(* CODESYS project TcMatrix.library
   DefaultNamespace: TcMatrix
   Description: Matrix arithmatic library
   Author: Andrew Burks
   DocFormat: reStructuredText
   Title: TcMatrix
   Version: 1.4.3
   Company: Burks Engineering
   Placeholder: TcMatrix

Project tree, tasks and I/O mapping:
  libraries: Tc2_Standard, * (Beckhoff Automation GmbH); Tc2_System, * (Beckhoff Automation GmbH); Tc2_Utilities, * (Beckhoff Automation GmbH); Tc3_DynamicMemory, * (Beckhoff Automation GmbH)
  POUs/
    Csv/
      function block MatrixCsvReader [ST]
      function block MatrixCsvWriter [ST]
    Functions/
      Arrays/
        function Array2D_Cols [ST]
        function Array2D_Rows [ST]
        function Array2D_To_Matrix [ST]
        function Matrix_SameSizeAs_Array2D [ST]
        function Matrix_To_Array2D [ST]
      Matrix/
        function Matrix_CanMult [ST]
        function Matrix_Copy [ST]
        function Matrix_DeterminateSquare [ST]
        function Matrix_ElementDifference [ST]
        function Matrix_ElementProduct [ST]
        function Matrix_ElementSum [ST]
        function Matrix_Grow [ST]
        function Matrix_InvertSquare [ST]
        function Matrix_Product [ST]
        function Matrix_Scale [ST]
        function Matrix_Shrink [ST]
        function Matrix_SubMatrix [ST]
        function Matrix_Transpose [ST]
        function Matrix_TransposeSquare [ST]
      Vector/
        function Vector_CrossProduct [ST]
        function Vector_DotProduct [ST]
        function Vector_Magnitude [ST]
        function Vector_Normalize [ST]
    MatrixAccessors/
      function block MatrixAccessor [ST]: Init_, This2Parent, GetI, SetI
      function block ShrunkMatrixAccessor [ST]: Init, Cols, Rows, This2Parent
      function block SubMatrixAccessor [ST]: Init, Cols, Rows, This2Parent
      function block TransposeMatrixAccessor [ST]: Init, Cols, Rows, This2Parent
    function block Array2DStaticMatrix [ST]: GetI, SetI
    function block DynamicMatrix [ST]: LogData, Free, Init, InitArray2D, InitConstant, InitCopy, InitIdentity, InitMagicSquare, InitTrapezoidal, InitVector, InitZeros, Grow, Resize, Shrink, Transpose, Cols, FB_exit, FB_init, GetI, Rows, SetI, AsColVector, AsElementDifference, AsElementProduct, AsElementSum, AsGrown, AsInverse, AsMatrixProduct, AsRowVector, AsScaled, AsShrunk, AsSubMatrix, AsTransposed, AsVectorCrossProduct
    function block ExternalStaticMatrix [ST]: Init, GetI, SetI
    function block Matrix [ST]: GetShrunkMatrixAccessor, GetSubMatrixAccessor, GetTransposeMatrixAccessor, Average, MaxVal, MinVal, Sum, IsEqual, IsEqualSize, IsNearlyEqual, GetDeterminant, GetI, GetRC, GetSize, GetVectorDotProduct, GetVectorMagnitude, CopyTo, GetStringLengthEstimate, IsCleared, IsEmpty, IsNearZero, IsSquare, IsVector, LogError, LogEvent, LogMessage, LogWarning, WriteDataToString, Clear, CopyFrom, ElementDifference, ElementProduct, ElementSum, FillFrom, FillFromArray2D, FillFromAt, FillTrapezoidal, IntPower, InvertSquare, Normalize, Power, Scale, SetI, SetRC, SortByColAsc, SwapI, SwapRC, SwapRow, TransposeSquare, BufferSize, Cols, Length, Rows, sPath, ZeroReference, IC2RC, RC2I, RCC2I
    function block StaticMatrix [ST]: Init_, Cols, Rows
  Version/
    global variables Global_Version
*)

// Version/Global_Version
{attribute 'TcGenerated'}
{attribute 'no-analysis'}
{attribute 'linkalways'}
// This function has been automatically generated from the project information.
VAR_GLOBAL CONSTANT
	{attribute 'const_non_replaced'}
	stLibVersion_TcMatrix : ST_LibVersion := (iMajor := 1, iMinor := 4, iBuild := 3, iRevision := 0, nFlags := 0, sVersion := '1.4.3');
END_VAR

// POUs/Csv/MatrixCsvReader
FUNCTION_BLOCK MatrixCsvReader
VAR_IN_OUT CONSTANT
	M : Matrix;
END_VAR
VAR_INPUT
	bExecute : BOOL;
	sPathName : T_MaxString;
	tTimeout : TIME;//timeout applied indidivudally to each file operation
	nHeaderLines : UDINT;//number of lines to skip at the beginning
END_VAR
VAR_OUTPUT
	bBusy : BOOL;
	bError : BOOL;
	nErrId : UDINT;
	nErrStep : UDINT;
	nRows : UINT;
	nCols : UINT;
	nVals : UINT;
END_VAR
VAR
	FileOpen : FB_FileOpen;
	CsvRead : FB_CSVMemBufferReader;
	FileRead : FB_FileRead;
	FileSeek : FB_FileSeek;
	FileClose : FB_FileClose;
	
	hFile : UINT;
	readEOF : BOOL;
	bytesRead : DINT;
	bytesParsed : DINT;
	buffer : STRING(bufferSize);
	step : UDINT;
	
	Hi : UINT;
	Ri : UINT;
	Ci : UINT;
	BuffCmd : E_EnumCmdType;
END_VAR
VAR CONSTANT
	bufferSize : UDINT := 1024;
	dataSize : UDINT := 16;	

	stepReady : UDINT := 0;
	stepOpenFile : UDINT := 1;
	stepFillBuffer : UDINT := 2;
	stepReadBuffer : UDINT := 3;
	stepMovePointer : UDINT := 4;
	stepCloseFile : UDINT := 5;
	stepDone : UDINT := 6;
END_VAR

FileOpen(
	sNetId := '',
	sPathName := spathname,
	nMode := FOPEN_MODEREAD OR FOPEN_MODEBINARY,
	ePath := E_OpenPath.PATH_GENERIC,
	bExecute := step = stepOpenFile,
	tTimeout := tTimeout);
FileRead(snetId := '',
	hFile := hFile,
	pReadBuff := ADR(buffer),
	cbReadLen := bufferSize,
	bExecute := step = stepFillBuffer,
	tTimeout := tTimeout);
FileSeek(snetID := '',
	hFile := hFile,
	//nSeekPos := 0,
	eOrigin := E_SeekOrigin.SEEK_CUR,
	bExecute := step = stepMovePointer,
	tTimeout := tTimeout);
FileClose(
	snetId := '',
	hFile := hFile,
	bexecute := step = stepCloseFile,
	tTimeout := tTimeout);
			
CASE step OF
	stepReady:
		bError := FALSE;
		nErrId := 0;
		nErrStep := 0;
		
		hFile := 0;
		readEOF := FALSE;
		
		Hi := 0;
		Ri := 0;
		Ci := 0;
		nRows := 0;
		nCols := 0;
		
		IF bExecute THEN
			IF NOT M.IsEmpty THEN
				bBusy := TRUE;
				step := stepOpenFile;
			END_IF
		END_IF
		
	stepOpenFile:
		
		IF FileOpen.bError THEN
			bError := TRUE;
			nErrId := FileOpen.nErrId;
			nErrStep := step;
			step := stepDone;
		ELSIF NOT(FileOpen.bBusy) THEN
			hFile := FileOpen.hFile;
			step := stepFillBuffer;
		END_IF
		
	stepFillBuffer:
		bytesRead := 0;
		IF FileRead.bError THEN
			bError := TRUE;
			nErrId := FileRead.nErrId;
			nErrStep := step;
			step := stepCloseFile;
		ELSIF NOT(FileRead.bBusy) THEN
			bytesRead := UDINT_TO_DINT(FileRead.cbRead);
			readEOF := FileRead.bEOF;//it looks like EOF is mutually exclusive with actually reading bytes. so kind of useless.
			IF bytesRead = 0 THEN
				step := stepCloseFile;
			ELSE
				step := stepReadBuffer;
			END_IF
		END_IF
		
	stepReadBuffer:
		BuffCmd := E_EnumCmdType.eEnumCmd_First;
		bytesParsed := 0;
		REPEAT
			CsvRead(eCmd := BuffCmd,
				pBuffer := ADR(Buffer),
				cbBuffer := DINT_TO_UDINT(bytesRead));
			BuffCmd := E_EnumCmdType.eEnumCmd_Next;
			
			IF CsvRead.bOk THEN
				bytesparsed := bytesparsed + UDINT_TO_DINT(CsvRead.cbRead);
				IF Hi < nHeaderLines THEN
					IF CsvRead.bCRLF THEN
						Hi := Hi + 1;
					END_IF
				ELSE
					IF Ri >= M.Rows OR Ci >= M.Cols THEN
						bError := TRUE;
						nErrId :=1;
						nErrStep := step;
						step := stepCloseFile;
						RETURN;
					END_IF
					M.SetRC(Ri,Ci,STRING_TO_LREAL(CsvRead.getValue));
					Ci := Ci + 1;
					nVals := NVals + 1;
					IF CsvRead.bCRLF THEN
						Ri := Ri + 1;
						Ci := 0;
						nRows := Ri;
					END_IF
					IF Ci > nCols THEN
						nCols := Ci;
					END_IF
				END_IF
			END_IF
		UNTIL
			NOT(CsvRead.bOk)
		END_REPEAT
		IF readEOF THEN//this probably will never happen because EOF seems to be mutually exclusive with reading bytes
			step := stepCloseFile;
		ELSE
			//move pointer backwards to where it was before the read, then forward based on how much data was read from the CSV buffer. This re-reads any partial cells that were not parsed
			FileSeek.nSeekPos := bytesParsed - bytesRead;
			IF FileSeek.nSeekPos <> 0 THEN
				step := stepMovePointer;
			ELSE
				step := stepFillBuffer;
			END_IF;
		END_IF
		
	
		
	stepMovePointer:
		IF FileSeek.bError AND NOT bError THEN
			bError := TRUE;
			nErrId := FileSeek.nErrId;
			nErrStep := step;
			step := stepDone;
		ELSIF NOT(FileSeek.bBusy) THEN
			step := stepFillBuffer;
		END_IF
		
	stepCloseFile:
		
		IF FileClose.bError AND NOT bError THEN
			bError := TRUE;
			nErrId := FileClose.nErrId;
			nErrStep := step;
			step := stepDone;
		ELSIF NOT(FileClose.bBusy) THEN
			step := stepDone;
		END_IF
		
		
	stepDone:
		bBusy := FALSE;
END_CASE

IF NOT bExecute THEN
	step := stepReady;
	bBusy := FALSE;
END_IF

END_FUNCTION_BLOCK

// POUs/Matrix
(*
Matrix Base Class
=============

Overview
-------------

This abstract class encapsulates the logic of manipulating and interacting with matricies without forcing a specific memory management pattern.
Derived classes are:

- DynamicMatrix: A concrete class that dynamically allocates memory to take any form needed
- StaticMatrix: An abstract class that serves as the base for classes with fixed memory sources
- MatrixAccessor: An abstract class that serves as the base for classes that inherit the memory of another matrix and remap it to their own form
 
With either pattern the memory is accessed as a row-major 1D array of LREAL.

*)
{attribute 'reflection'}
{attribute 'no_assign'}
FUNCTION_BLOCK ABSTRACT Matrix
VAR_INPUT
END_VAR
VAR_OUTPUT
END_VAR
VAR

	
	{attribute 'instance-path'}
	{attribute 'noinit'}
	sPath_ : T_MaxString;
	
	Ri : UINT;
	Ci : UINT;
	I : UINT;
	
	ZeroReference_ : LREAL;//numbers below this are considered zero for the purposes of avoiding near-divide-by-zero floating point issues
END_VAR

LogMessage('%s: There is no need to call the main FB function for type Matrix');

METHOD PUBLIC GetShrunkMatrixAccessor : ShrunkMatrixAccessor
VAR_INPUT
	Row : UINT;
	Col : UINT;
END_VAR
GetShrunkMatrixAccessor.Init(THIS^,Row,Col);
END_METHOD

METHOD PUBLIC GetSubMatrixAccessor : SubMatrixAccessor
VAR_INPUT
	RowStart : UINT;
	RowCount : UINT;
	ColStart : UINT;
	ColCount : UINT;
END_VAR
GetSubMatrixAccessor.Init(THIS^,RowStart,RowCount,ColStart,ColCount);
END_METHOD

METHOD PUBLIC GetTransposeMatrixAccessor : TransposeMatrixAccessor
VAR_INPUT
END_VAR
GetTransposeMatrixAccessor.Init(THIS^);
END_METHOD

//returns the average value of all elements
PROPERTY PUBLIC Average : LREAL
GET
IF Length > 0 THEN
	Average := Sum / Length;
ELSE
	Average := 0;
END_IF
END_GET
END_PROPERTY

//Returns the maximum value from all elements
PROPERTY PUBLIC MaxVal : LREAL
GET
VAR
	MaxVal_ : LREAL;
END_VAR
IF IsEmpty THEN
	MaxVal := 0;
ELSE
	MaxVal_ := GetI(0);
	FOR I := 1 TO Length-1 DO
		IF getI(I) < MaxVal_ THEN
			MaxVal_ := GetI(I);
		END_IF
	END_FOR
	MaxVal := MaxVal_;
END_IF
END_GET
END_PROPERTY

//Returns the minimum value from all elements
PROPERTY PUBLIC MinVal : LREAL
GET
VAR
	MinVal_ : LREAL;
END_VAR
IF IsEmpty THEN
	MinVal := 0;
ELSE
	MinVal_ := GetI(0);
	FOR I := 1 TO Length-1 DO
		IF getI(I) < MinVal_ THEN
			MinVal_ := GetI(I);
		END_IF
	END_FOR
	MinVal := MinVal_;
END_IF
END_GET
END_PROPERTY

//Returns the sum of all elements
PROPERTY PUBLIC Sum : LREAL
GET
VAR
	Sum_ : LREAL;
END_VAR
Sum_ := 0;
IF NOT(IsEmpty) THEN
	FOR I := 0 TO Length-1 DO
		Sum_ := Sum_ + GetI(I);
	END_FOR
END_IF
Sum := Sum_;
END_GET
END_PROPERTY

//Determines if this matrix is equal to a supplied matrix.
//
//Two matricies are considered equal if they are the same size and every set of corresponding elements are equal.
//
//.. note:: Two empty matricies are considered equal.
METHOD PUBLIC IsEqual : BOOL//TRUE if the two matricies are equal, FALSE if they are not
VAR_IN_OUT CONSTANT
	M : Matrix;//The other matrix to compare to this one
END_VAR
IF NOT( IsEqualSize(M)) THEN
	IsEqual := FALSE;
	RETURN;
END_IF

//If either matrix is empty don't bother comparing elements
IF IsEmpty OR M.IsEmpty THEN
	//If both are empty then they are equal
	IsEqual := IsEmpty AND M.IsEmpty;
	RETURN;
END_IF

//Both Rows and Cols must be non zero for this loop to not go bonkers
FOR Ri := 0 TO Rows-1 DO
	FOR Ci := 0 TO Cols-1 DO
		IF NOT(GetRC(Ri,Ci) = M.GetRC(Ri,Ci)) THEN
			IsEqual := FALSE;
			RETURN;
		END_IF
	END_FOR
END_FOR

IsEqual := TRUE;
END_METHOD

//Checks if this matrix is the same size (number of rows and number of columns match) as the supplied matrix.
//
//.. note:: two empty matricies are considered the same size.
METHOD PUBLIC IsEqualSize : BOOL//True if this matrix is the same size as the supplied matrix
VAR_IN_OUT CONSTANT
	M : Matrix;//The matrix which should have its size compared to the size of this matrix
END_VAR
IsEqualSize := M.Rows = Rows AND M.Cols = Cols;
END_METHOD

//Determines if this matrix is *nearly* equal to a supplied matrix, based on a supplied precision.
//
//Two matricies are considered nearly equal if they are the same size and every set of corresponding elements are equal to within the supplied precision.
//.. note:: Note that two empty matricies are considered equal
METHOD PUBLIC IsNearlyEqual : BOOL//TRUE if the two matricies are nearly equal, FALSE if they are not
VAR_IN_OUT CONSTANT
	M : Matrix;//The other matrix to compare to this one
END_VAR
VAR_INPUT
	Precision : LREAL;//Deviation between two elements larger than this value makes them unequal
END_VAR
IF NOT( IsEqualSize(M)) THEN
	IsNearlyEqual := FALSE;
	RETURN;
END_IF

//If either matrix is empty don't bother comparing elements
IF IsEmpty OR M.IsEmpty THEN
	//If both are empty then they are equal
	IsNearlyEqual := IsEmpty AND M.IsEmpty;
	RETURN;
END_IF

//Both Rows and Cols must be non zero for this loop to not go bonkers
FOR Ri := 0 TO Rows-1 DO
	FOR Ci := 0 TO Cols-1 DO
		IF NOT( ABS(GetRC(Ri,Ci) - M.GetRC(Ri,Ci)) < Precision) THEN
			IsNearlyEqual := FALSE;
			RETURN;
		END_IF
	END_FOR
END_FOR

IsNearlyEqual := TRUE;
END_METHOD

//Gets the determinant of this matrix
//
//:Prerequisites:
// - Matrix is not empty
// - Matrix is square
//
//.. note:: If this matrix does not meet the requirements 0 is returned
METHOD PUBLIC GetDeterminant : LREAL//The determinant of this matrix, if the prerequisites are met. Otherwise, returns 0.
VAR_INPUT
END_VAR
VAR
	Res : LREAL;
END_VAR
IF NOT(Matrix_DeterminateSquare(M := THIS^,Res => Res)) THEN
	LogWarning('%s: Unable to calculate determinate');
	GetDeterminant := 0;
ELSE
	GetDeterminant := Res;
END_IF
END_METHOD

//Gets the value of the element in this matrix at the supplied location as if the elements were stored in a 1D row-major array
//
//:Prerequisites:
// - I < Rows*Cols
// - Matrix is not empty
//
//.. note:: If the supplied index is out of bounds the value 0 is returned and a warning is generated in the Error List
METHOD PUBLIC ABSTRACT GetI : LREAL//The value of the element at the specified index, or 0 if an invalid index is supplied
VAR_INPUT
	I : UINT;//The index of the element which should have its value returned
END_VAR
END_METHOD

//returns the value of the element of this matrix at the specified row and column.
//
//:Prerequisites:
// - Row < Rows
// - Col < Cols
// - Matrix is not empty
//
//.. note:: If the supplied or or column is out of bounds then a warning message is generated in the Error List and the value 0 is returned
METHOD PUBLIC GetRC : LREAL//The value of the element at the specified row and column, or 0 if an invalid index is supplied
VAR_INPUT
	Row : UINT;//The row of the element to fetch
	Col : UINT;//The column of the element to fetch
END_VAR
IF IsEmpty THEN
	GetRC := 0;
	LogWarning('%s: Attempted RC access of empty Matrix');
ELSIF
	Row >= Rows THEN
	GetRC := 0;
	LogWarning('%s: Attempted RC access of out-of-bound matrix row');
ELSIF
	Col >= Cols THEN
	GetRC := 0;
	LogWarning('%s: Attempted RC access of out-of-bounds Matrix column');
ELSE
	GetRC := GetI(RC2I(Row,Col));
END_IF
END_METHOD

//Returns the length of the matrix in the specified dimension
//
// - GetSize(0) is equivalent to Rows
// - GetSize(1) is equivalent to Cols
//
//.. note:: If an invalid dimension is supplied then a warning is generated in the Error List and the value 0 is returned
METHOD PUBLIC GetSize : UINT//The length of the matrix in the specified dimension, or 0 if the dimension specified is invalid
VAR_INPUT
	Dim : UINT;//The dimension of the matrix for which the size should be returned. 0=Rows, 1=Cols
END_VAR
IF Dim = 0 THEN
	GetSize := Rows;
ELSIF Dim = 1 THEN
	GetSize := Cols;
ELSE
	LogWarning('%s: Attempted to GetSize for a dimension other than 0 or 1');
	GetSize := 0;
END_IF
END_METHOD

//Returns the vector dot product of this matrix and the supplied other matrix (ignoring the orientation of both matricies).
//:Prerequisites:
// - This matrix is a vector and is not empty
// - The supplied other matrix is a vector and is not empty
// - This vector has the same length (but not necessarily orientation) as the supplied vector
METHOD PUBLIC GetVectorDotProduct : LREAL//The dot product (element-wise product) of this vector and the supplied vector, or 0 if the inputs are invalid
VAR_IN_OUT CONSTANT
	V : Matrix;//The vector which which the dot product of this vector should be taken.
END_VAR
VAR
	Res : LREAL;
END_VAR
IF NOT(Vector_DotProduct(V,THIS^,Res => Res)) THEN
	LogWarning('%s: Unable to calculate vector dot product');
	GetVectorDotProduct := 0;
ELSE
	GetVectorDotProduct := Res;
END_IF
END_METHOD

//Calcualtes the vector magnitude of this matrix (square root of the sum of the squares), assuming it is a vector.
//
//:Prerequisites:
// - This matrix is not empty and is a vector
//
//.. note:: If this matrix is empty or is not a vector, 0 is returned
METHOD PUBLIC GetVectorMagnitude : LREAL//The vector magnitude of this matrix if it is a vector, otherwise 0
VAR_INPUT
END_VAR
VAR
	Res : LREAL;
END_VAR
IF NOT(Vector_Magnitude(THIS^,Res => Res)) THEN
	LogWarning('%s: Unable to calculate vector magnitude');
	GetVectorMagnitude := 0;
ELSE
	GetVectorMagnitude := Res;
END_IF
END_METHOD

(*Copy the value from each element in this matrix to each corresponding element in the destination matrix

:Prerequisites:
 - This matrix is the same size as the destination matrix
 - Neither matrix is empty
 
 *)
METHOD PUBLIC CopyTo : BOOL//Returns true if the prerequisites were met and the data was copied, false otherwise
VAR_IN_OUT
	M : Matrix;//Destination for the copy operation
END_VAR
CopyTo := Matrix_Copy(THIS^,M);
END_METHOD

//Calulates how long of a string (in Bytes) is required in order to print the entire contents of the matrix using the WriteDataToString function
METHOD PUBLIC GetStringLengthEstimate : UDINT;
VAR_INPUT
END_VAR
VAR
	CharsPerElement : UDINT := 20;//15 point precision, decimal, sign, leading zero, comma, space
	CharsPerRow : UDINT := 6;//space, semicolon, carriage return, line return, space, space
	CharsPerMatrix : UDINT := 4;//open bracket, space ; space, closing bracket
END_VAR
GetStringLengthEstimate := 1+CharsPerMatrix + CharsPerRow * Rows + CharsPerElement * Length;//extra one for null character
END_METHOD

//Returns TRUE if every element of the matrix is equal to zero, or the matrix is empty
PROPERTY PUBLIC IsCleared : BOOL
GET
IF IsEmpty THEN
	IsCleared := TRUE;
	RETURN;
END_IF

FOR Ri := 0 TO Rows-1 DO
	FOR Ci := 0 TO Cols-1 DO
		IF GetRC(Ri,Ci) <> 0 THEN
			IsCleared := FALSE;
			RETURN;
		END_IF
	END_FOR
END_FOR

IsCleared := TRUE;
END_GET
END_PROPERTY

//Returns true if the matrix does not have any addresible elements
PROPERTY PUBLIC IsEmpty : Bool
GET
IsEmpty := Length = 0;
END_GET
END_PROPERTY

//Returns true if the supplied value is near enough to zero that it should not be used as a divisor. See the property ZeroReference
METHOD PROTECTED IsNearZero : BOOL
VAR_INPUT
	IN : LREAL;//The value which should have its magnitude evaluated
END_VAR
IsNearZero := ABS(IN) < ZeroReference;
END_METHOD

//Returns true if this matrix is not empty, and the number of columns is equal to the number of rows
PROPERTY PUBLIC IsSquare : BOOL
GET
IsSquare := NOT(IsEmpty) AND Rows = Cols;
END_GET
END_PROPERTY

//Returns true if this matrix is not empty, and at least one dimension has a size of 1 (row vector or column vector).
PROPERTY PUBLIC IsVector : BOOL
GET
IsVector := NOT(IsEmpty) AND (Rows = 1) OR (Cols = 1);
END_GET
END_PROPERTY

//Logs the supplied message to the error output as an 'Error'
METHOD PROTECTED LogError
VAR_INPUT
	Message : T_MaxString;//The message to log. %s is substituted with the symbolic address of this matrix.
END_VAR
ADSLOGSTR(ADSLOG_MSGTYPE_WARN,Message,sPath);
END_METHOD

//Logs the supplied message to the windoes event log
METHOD PROTECTED LogEvent
VAR_INPUT
	Message : T_MaxString;//The message to log. %s is substituted with the symbolic address of this matrix.
END_VAR
ADSLOGSTR(ADSLOG_MSGTYPE_LOG,Message,sPath);
END_METHOD

//Logs the supplied message to the error output as a 'Message'
METHOD PROTECTED LogMessage
VAR_INPUT
	Message : T_MaxString;//The message to log. %s is substituted with the symbolic address of this matrix.
END_VAR
ADSLOGSTR(ADSLOG_MSGTYPE_STRING,Message,sPath);
END_METHOD

//Logs the supplied message to the error output as a 'Warning'
METHOD PROTECTED LogWarning
VAR_INPUT
	Message : T_MaxString;//The message to log. %s is substituted with the symbolic address of this matrix.
END_VAR
ADSLOGSTR(ADSLOG_MSGTYPE_WARN,Message,sPath);
END_METHOD

//Writes the elements of this matrix to a string in a human-readable way, up to the specified length.
//
//Use the GetStringLengthEstimate function to calculate how much memory is necessary to output the entire matrix to one string
METHOD PUBLIC WriteDataToString : BOOL//Returns true if the entire matrix was written to the string, false otherwise
VAR_INPUT
	Buffer : POINTER TO STRING;//The output buffer that should be overwritten with the contents of the matrix
	BufferLen : UDINT;//The length, in bytes, of the output buffer available fo writing
END_VAR
VAR
	Temp : STRING(32);
	Pos : UDINT;
END_VAR
VAR CONSTANT
	ColSep : STRING(2) := ', ';
	RowSep : STRING(6) := ' ;$R$L  ';
	MatStart : STRING(2) := '[ ';
	MatEnd : STRING(2) := ' ]';
END_VAR
Pos := 0;
IF NOT(STRNCPY(Buffer+Pos,ADR(MatStart),BufferLen-Pos)) THEN
	WriteDataToString := FALSE;
	RETURN;
END_IF;
Pos := Pos + LEN2(ADR(MatStart));

FOR Ri := 0 TO Rows-1 DO
	IF Ri <> 0 THEN
		IF NOT(STRNCPY(Buffer+Pos,ADR(RowSep),BufferLen-Pos)) THEN
			WriteDataToString := FALSE;
			RETURN;
		END_IF;
		Pos := Pos + LEN2(ADR(RowSep));
	END_IF;

	FOR Ci := 0 TO Cols-1 DO
		IF Ci <> 0 THEN
			IF NOT(STRNCPY(Buffer+Pos,ADR(ColSep),BufferLen-Pos)) THEN
				WriteDataToString := FALSE;
				RETURN;
			END_IF;
			Pos := Pos + LEN2(ADR(ColSep));
		END_IF;
		
		Temp := LREAL_TO_STRING(GetRC(Ri,Ci));
		IF NOT(STRNCPY(Buffer+Pos,ADR(Temp),BufferLen-Pos)) THEN
			WriteDataToString := FALSE;
			RETURN;
		END_IF;
		Pos := Pos + LEN2(ADR(Temp));
	END_FOR
END_FOR

IF NOT(STRNCPY(Buffer+Pos,ADR(MatEnd),BufferLen-Pos)) THEN
	WriteDataToString := FALSE;
	RETURN;
END_IF;
Pos := Pos + LEN2(ADR(MatEnd));
WriteDataToString := TRUE;
END_METHOD

//Resets the value of every element in this matrix to zero
METHOD PUBLIC Clear
VAR_INPUT
END_VAR
FillTrapezoidal(0,0,0);
END_METHOD

(*Copy the value from each element in the source matrix to each corresponding element in this matrix

:Prerequisites:
 - This matrix is the same size as the source matrix
 - Neither matrix is empty
 
 *)
METHOD PUBLIC CopyFrom : BOOL//Returns true if the prerequisites were met and the data was copied, false otherwise
VAR_IN_OUT CONSTANT
	M : Matrix;//Source of the copy operation
END_VAR
CopyFrom := Matrix_Copy(M_From := M, M_To := THIS^);
END_METHOD

(*
For each element in this matrix, calculate a new value by Subtracting the value of the corresponding element of the supplied matrix from the value in this matrix

THIS := THIS - M

:Prerequisites:
 - This matrix is the same size as the supplied matrix
 - Neither matrix is empty
 
 *)
METHOD PUBLIC ElementDifference : BOOL//TRUE if the operation completes successfully, false if the prerequisites are not met
VAR_IN_OUT CONSTANT
	M : Matrix;//the subtrahend in the subtraction
END_VAR
ElementDifference := Matrix_ElementDifference(THIS^,M,THIS^);
END_METHOD

(*
For each element in this matrix, calculate a new value by Multiplying the value of the corresponding element of the supplied matrix with the value in this matrix

THIS := THIS .* M

:Prerequisites:
 - This matrix is the same size as the supplied matrix
 - Neither matrix is empty
 
 *)
METHOD PUBLIC ElementProduct : BOOL//TRUE if the operation completes successfully, false if the prerequisites are not met
VAR_IN_OUT CONSTANT
	M : Matrix;//the supplied matrix to be multiplied element-by-element to this matrix
END_VAR
ElementProduct := Matrix_ElementProduct(THIS^,M,THIS^);
END_METHOD

(*
For each element in this matrix, calculate a new value by Adding the value of the corresponding element of the supplied matrix with the value in this matrix

THIS := THIS + M

:Prerequisites:
 - This matrix is the same size as the supplied matrix
 - Neither matrix is empty
 
 *)
METHOD PUBLIC ElementSum : BOOL//TRUE if the operation completes successfully, false if the prerequisites are not met
VAR_IN_OUT CONSTANT
	M : Matrix;//the supplied matrix to be added to this matrix
END_VAR
ElementSum := Matrix_ElementSum(THIS^,M,THIS^);
END_METHOD

(*
For every element that exist in both this matrix and the source matrix, copy the value from the source matrix into this matrix
*)
METHOD PUBLIC FillFrom
VAR_IN_OUT CONSTANT
	M : Matrix;//source matrix for element copy operation
END_VAR
IF M.IsEmpty OR IsEmpty THEN
	RETURN;//no need to fill to/from empty matricies, and it
END_IF

FOR Ri := 0 TO MIN(Rows,M.Rows)-1 DO
	FOR Ci := 0 TO MIN(Cols,M.Cols)-1 DO
		SetRC(Ri,Ci,M.GetRC(Ri,Ci));
	END_FOR
END_FOR
END_METHOD

(*
For every element that exist in both this matrix and the source array, copy the value from the source array into this matrix
*)
METHOD PUBLIC FillFromArray2D
VAR_IN_OUT CONSTANT
	A : ARRAY[*,*] OF LREAL;//source matrix for element copy operation
END_VAR
VAR
	inRows : UINT;
	inCols : UINT;
END_VAR
IF LOWER_BOUND(A,1) < UPPER_BOUND(A,1) OR LOWER_BOUND(A,2) < UPPER_BOUND(A,2)  OR IsEmpty THEN
	RETURN;//no need to fill to/from empty matricies
END_IF

inRows := DINT_TO_UINT(UPPER_BOUND(A,1) - LOWER_BOUND(A,1) + 1);
inCols := DINT_TO_UINT(UPPER_BOUND(A,2) - LOWER_BOUND(A,2) + 1);

FOR Ri := 0 TO MIN(Rows,inRows)-1 DO
	FOR Ci := 0 TO MIN(Cols,inCols)-1 DO
		SetRC(Ri,Ci,A[LOWER_BOUND(A,1)+Ri,LOWER_BOUND(A,2)+Ci]);
	END_FOR
END_FOR
END_METHOD

//Consider the subset of elements in this matrix starting and the supplied initial row and column as a submatrix. 
//For every element that exists in both the submatrix and the supplies source matrix, copy the value from the source matrix into the corresponding element of the submatrix.
METHOD PUBLIC FillFromAt
VAR_IN_OUT CONSTANT
	M : Matrix;//Source matrix for the copy operation
END_VAR
VAR_INPUT
	RStart : UINT;//Row within this matrix to start the fill operation
	CStart : UINT;//Column within this matrix to start the fill operation
END_VAR

VAR
	SubMatrix : SubMatrixAccessor;
END_VAR
IF M.IsEmpty THEN
	LogWarning('%s: Attempt to fill from an empty matrix');
	RETURN;
END_IF

IF IsEmpty THEN
	LogWarning('%s: Attempt to fill into an empty matrix');
	RETURN;
END_IF

IF RStart >= Rows THEN
	LogWarning('%s: Attempt to fill out of bounds row of matrix');
	RETURN;
END_IF

IF CStart >= Cols THEN
	LogWarning('%s: Attempt to fill out of bounds col of matrix');
	RETURN;
END_IF

SubMatrix := GetSubMatrixAccessor(RStart,Rows-Rstart,CStart,Cols-CStart);
SubMatrix.FillFrom(M);
END_METHOD

//Fills all elements of this matrix based on which of three zones it is located into when considered as a trapezoidal matrix
METHOD PUBLIC FillTrapezoidal
VAR_INPUT
	Diagonal : LREAL;//Every element on the main diagonal of the matrix is set to this value.
	UpperRight : LREAL;//Every element above or to the right of the main diagonal is set to this value;
	LowerLeft : LREAL;//Every element below or to the left of the main diagonal is set to this value;
END_VAR
IF IsEmpty THEN
	LogWarning('%s: Attempt to trapezoid fill an empty matrix');
	RETURN;
END_IF


FOR Ri := 0 TO Rows-1 DO
	FOR Ci := 0 TO Cols-1 DO
		IF Ri = Ci THEN
			SetRC(Ri,Ci,Diagonal);
		ELSIF Ri < Ci THEN
			SetRC(Ri,Ci,UpperRight);
		ELSE
			SetRC(Ri,Ci,LowerLeft);
		END_IF
	END_FOR
END_FOR
END_METHOD

//Raises every element of the matrix to the supplied power
METHOD PUBLIC IntPower
VAR_INPUT
	Exponent : INT;//Power with which to raise every element of the matrix
END_VAR
IF IsEmpty THEN
	RETURN;
END_IF
FOR I := 0 TO Length-1 DO
	SetI(I,EXPT(GetI(I),Exponent));
END_FOR
END_METHOD

//Inverts the matrix. May fail if the matrix is too close to being singular. Use the tolerance input to specify how close to go (1E-6 to 1E-9 is porbably good).
//
//:Prerequisites:
//- This matrix is square
//- This matrix is not empty
METHOD PUBLIC InvertSquare : BOOL//True if the inverse has been calculated. False if a precondition was not met, or a near-singularity was detected (data may be malformed).
VAR_INPUT
	Tolerance : LREAL;//The smallest magnitude of number that is allowed to be used as a denominator in the calculation of the inverse
END_VAR
InvertSquare := Matrix_InvertSquare(THIS^,Tolerance);
END_METHOD

//Scales every element of the matrix by the inverse of the magnitude.
//
// - Vector magnitude is determined by GetVectorMagnitude
// - Square Matrix magnitude is determined by GetDeterminate
// - Rectangular matricies produce an error
//
//:Prerequisites: 
// - matrix is not empty
// - matrix is not rectangular
METHOD PUBLIC Normalize : BOOL//TRUE if the matrix was normalized. FALSE if not.
VAR_INPUT
END_VAR
VAR
	Mag : LREAL;
END_VAR
VAR CONSTANT
	
END_VAR
IF IsEmpty THEN
	Normalize := FALSE;
	LogWarning('%s: Unable to normalize matrix because it is empty');
	RETURN;
ELSIF IsVector THEN
	Mag := GetVectorMagnitude();
ELSIF IsSquare THEN
	Mag := GetDeterminant();
ELSE
	Normalize := FALSE;
	LogWarning('%s: Unable to normalize matrix because it is not square or a vector');
	RETURN;
END_IF

IF IsNearZero(Mag) THEN
	Normalize := FALSE;
	LogWarning('%s: Unable to normalize matrix because the magnitude was too close to zero');
	RETURN;
END_IF

Normalize := TRUE;

Scale(1/Mag);
END_METHOD

//Raises every element of the matrix to the supplied power
//
//.. caution:: Many values of exponent could easily cause all of the elements to turn into NaN!
METHOD PUBLIC Power
VAR_INPUT
	Exponent : LREAL;//Power with which to raise every element of the matrix
END_VAR
IF IsEmpty THEN
	RETURN;
END_IF
FOR I := 0 TO Length-1 DO
	SetI(I,EXPT(GetI(I),Exponent));
END_FOR
END_METHOD

//Scales every element of this matrix by the supplied value.
METHOD PUBLIC Scale
VAR_INPUT
	Scalar : LREAL;//Value with which to scale every element of this matrix
END_VAR
Matrix_Scale(THIS^,Scalar);
END_METHOD

//Sets the element specified by the supplied index to the suppleid value, assuming the data of the matrix is stored in a 1D row-major array
//
//:Prerequisites: - I < Rows*Cols
METHOD PUBLIC ABSTRACT SetI : BOOL//TRUE if the specified index is valid and the data is copied. FLASE otherwise
VAR_INPUT
	I : UINT;//The index specifying which element should be modified
	Val : LREAL;//The value copied to the corresponding element
END_VAR
END_METHOD

//Sets the element specified by the supplied row and column to the suppleid value
//
//:Prerequisites:
// - Row < Rows
// - Col < Cols
METHOD PUBLIC SetRC : BOOL;//TRUE if the specified row and column are valid and the data is copied. FALSE otherwise
VAR_INPUT
	Row : UINT;//The row of the element to set
	Col : UINT;//The column of the element to set
	Val : LREAL;//The value to copy into the specified element
END_VAR
IF IsEmpty THEN
	SetRC := FALSE;
	LogWarning('%s: Attempt to set data using RC access when data is not initialized');
ELSIF Row >= Rows THEN
	SetRC := FALSE;
	LogWarning('%s: Attempt to set data using RC access when Row is out of bounds');
ELSIF Col >= Cols THEN
	SetRC := FALSE;
	LogWarning('%s: Attempt to set data using RC access when Col is out of bounds');
ELSE
	SetRC := SetI(RC2I(Row,Col),Val);
END_IF
END_METHOD

//In-place bubble sort of rows by the specified col, into ascending order
//
//algorithm is 'stable', meaning that two equivalent rows will maintain their relative position after sorting.
//This is nice because it lets you sort by secondary/tertiary/etc columns (if you do them in reverse)
METHOD PUBLIC SortByColAsc : BOOL
VAR_INPUT
	SortCol : UINT;
END_VAR
VAR
	lastUnsortedRow : UINT;
	lastSwappedRow : UINT;
	Result : BOOL;
END_VAR
IF ISEmpty OR Rows <= 1 THEN
	SortByColAsc := FALSE;
	RETURN;
END_IF

lastUnsortedRow := Rows-1;
Result := TRUE;
REPEAT
	lastSwappedRow := 0;
	FOR Ri := 1 TO lastUnsortedRow DO
		IF GetRC(Ri-1,SortCol) >GetRC(Ri,SortCol) THEN
			Result := Result AND SwapRow(Ri-1,Ri);
			lastSwappedRow := Ri;
		END_IF
	END_FOR
	lastUnsortedRow := lastSwappedRow-1;
UNTIL
	lastSwappedRow = 0
END_REPEAT
END_METHOD

METHOD PUBLIC SwapI : BOOL
VAR_INPUT
	I1 : UINT;
	I2 : UINT;
END_VAR
VAR
	Temp : LREAL;
END_VAR
IF IsEmpty OR I1 >= Length OR I2 >= Length THEN
	SwapI := FALSE;
	RETURN;
END_IF
Temp := GetI(I1);
SwapI := SetI(I1,GetI(I2));
SwapI := SwapI AND SetI(I2,Temp);
END_METHOD

METHOD PUBLIC SwapRC : BOOL
VAR_INPUT
	R1 : UINT;
	C1 : UINT;
	R2 : UINT;
	C2 : UINT;
END_VAR
VAR
	Temp : LREAL;
END_VAR
IF IsEmpty OR R1 >= Rows OR R2 >= Rows OR C1 >= Cols OR C2 >= Cols THEN
	SwapRC := FALSE;
	RETURN;
END_IF
Temp := GetRC(R1,C1);
SwapRC := SetRC(R1,C1,GetRC(R2,C2));
SwapRC := SwapRC AND SetRC(R2,C2,Temp);
END_METHOD

METHOD PUBLIC SwapRow : BOOL
VAR_INPUT
	R1 : UINT;
	R2 : UINT;
END_VAR
VAR
	Result : BOOL;
END_VAR
IF IsEmpty OR R1 >= Rows OR R2 >= Rows THEN
	SwapRow := FALSE;
	RETURN;
END_IF


FOR Ci := 0 TO Cols-1 DO
	IF NOT(SwapRC(R1,Ci,R2,Ci)) THEN
		SwapRow := FALSE;
		RETURN;
	END_IF
END_FOR

SwapRow := TRUE;
END_METHOD

//Transposes the matrix.
//
//:Prerequisites:
//- This matrix is square
//- This matrix is not empty
METHOD PUBLIC TransposeSquare : BOOL//TRUE if the operation completes successfully, false if the prerequisites are not met
VAR_INPUT
END_VAR
VAR
	Temp : DynamicMatrix;
END_VAR
TransposeSquare := Matrix_TransposeSquare(THIS^);
END_METHOD

//The length (in Bytes) of the memory allocated to storing element data for this matrix
PROPERTY PUBLIC BufferSize : UDINT
GET
BufferSize := SIZEOF(LREAL)*Length;
END_GET
END_PROPERTY

//Total number of columns in this matrix
PROPERTY PUBLIC ABSTRACT Cols : UINT
GET
END_GET
END_PROPERTY

//Total number of elements in this matrix
PROPERTY PUBLIC Length : UINT
GET
Length := Rows * Cols;
END_GET
END_PROPERTY

//Total number of rows in this matrix
PROPERTY PUBLIC ABSTRACT Rows : UINT
GET
END_GET
END_PROPERTY

//The symbolic path to this matrix in memory
PROPERTY PUBLIC sPath : T_MaxString
GET
sPath := sPath_;
END_GET
END_PROPERTY

//Values with a magnitude lower than this value will be considered as zero for purposes of avoiding divide by zero errors
PROPERTY PUBLIC ZeroReference : LREAL
GET
ZeroReference := ZeroReference_;
END_GET
SET
ZeroReference_ := ZeroReference;
END_SET
END_PROPERTY

METHOD PROTECTED IC2RC
VAR_INPUT
	Index : UINT;
	ColCount : UINT;
END_VAR
VAR_OUTPUT
	Row : UINT;
	Col : UINT;
END_VAR
Col := Index MOD ColCount;
Row := (Index - Col) / ColCount;
END_METHOD

//Computes the index in a row-major 1D array representing this Matrix given a supplied Row and Column index
METHOD PROTECTED RC2I : UINT//The 0-based index of the element in the 1D array
VAR_INPUT
	Row : UINT;//The target row of the element
	Col : UINT;//The target column of the element
END_VAR
RC2I := RCC2I(Row,Col,Cols);
END_METHOD

//Computes the index in a row-major 1D array representing a Matrix with the supplied number of columns (*NOT this matrix*) given a supplied Row and Column index
METHOD PROTECTED RCC2I : UINT//Index of the element in a 1D array
VAR_INPUT
	Row : UINT;//Row of the target element
	Col : UINT;//Column fo the target element
	ColCount : UINT;//The number of columns in the 1D array (not necessarilly the number of columns in this Matrix!)
END_VAR
RCC2I := Row*ColCount + Col;
END_METHOD

END_FUNCTION_BLOCK

// POUs/DynamicMatrix
{attribute 'no_assign'}
{attribute 'reflection'}
FUNCTION_BLOCK DynamicMatrix EXTENDS Matrix
VAR_INPUT
END_VAR
VAR_OUTPUT
END_VAR
VAR
	Rows_ : UINT := 0;
	Cols_ : UINT := 0;
	
	Data : POINTER TO LREAL;//1D array of reals, such that I = F(R,C) = R*Cols + C (row-major)
	
	MemManager : FB_DynMem_Manager2;
END_VAR

METHOD PUBLIC LogData : BOOL
VAR_INPUT
	Message : T_MaxString;
END_VAR
VAR
	BufferLen : UDINT;
	Buffer : POINTER TO STRING;
END_VAR
BufferLen := GetStringLengthEstimate();
Buffer := MemManager.Alloc(BufferLen+INT_TO_UDINT(Len(Message))+2,FALSE);
IF Buffer = 0 THEN
	LogData := FALSE;
	RETURN;
END_IF
Buffer^ := CONCAT(Message,'$R$L');//writes null character to first element?
IF NOT(WriteDataToString(Buffer+INT_TO_DWORD(LEN(Message))+2,BufferLen)) THEN
	LogData := FALSE;
	MemManager.Free2(Buffer);
	RETURN;
END_IF
ADSLOGSTR(ADSLOG_MSGTYPE_LOG OR ADSLOG_MSGTYPE_STRING, Buffer^,sPath);
MemManager.Free2(Buffer);
END_METHOD

METHOD PUBLIC Free
VAR_INPUT
END_VAR
Resize(0,0,FALSE,FALSE);
Rows_ := 0;
Cols_ := 0;
IF Data <> 0 THEN
	MemManager.Free2(Data);
END_IF;
END_METHOD

METHOD PUBLIC Init : BOOL
VAR_INPUT
	Rows : UINT;
	Cols : UINT;
END_VAR
Init := Resize(Rows,Cols,FALSE,FALSE);
END_METHOD

METHOD PUBLIC InitArray2D : BOOL
VAR_IN_OUT CONSTANT
	A : ARRAY[*,*] OF LREAL;
END_VAR
VAR
	inRows : UINT;
	inCols : UINT;
END_VAR
inRows := DINT_TO_UINT(UPPER_BOUND(A,1) - LOWER_BOUND(A,1) + 1);
inCols := DINT_TO_UINT(UPPER_BOUND(A,2) - LOWER_BOUND(A,2) + 1);

IF NOT(Init(inRows,inCols)) THEN
	InitArray2D := FALSE;
	RETURN;
END_IF

InitArray2D := Array2D_To_Matrix(A,THIS^);
END_METHOD

METHOD PUBLIC InitConstant : BOOL;
VAR_INPUT
	Rows : UINT;
	Cols : UINT;
	Val : LREAL;
END_VAR
InitConstant := InitTrapezoidal(Rows,Cols,Val,Val,Val);
END_METHOD

METHOD PUBLIC InitCopy : BOOL
VAR_IN_OUT CONSTANT
	M : Matrix;
END_VAR
IF NOT(Init(M.Rows,M.Cols)) THEN
	InitCopy := FALSE;
	RETURN;
END_IF

InitCopy := TRUE;

FillFrom(M);
END_METHOD

METHOD PUBLIC InitIdentity : BOOL;
VAR_INPUT
	Size : UINT;
END_VAR
InitIdentity := InitTrapezoidal(Size,Size,1,0,0);
END_METHOD

METHOD PUBLIC InitMagicSquare : BOOL
VAR_INPUT
	Size : UINT;//must be an odd number!
END_VAR
VAR 
	Result : BOOL;	
END_VAR
//source: https://en.wikipedia.org/wiki/Magic_square#A_method_for_constructing_a_magic_square_of_odd_order

IF Size MOD 2 = 0 THEN
	InitMagicSquare := FALSE;
	RETURN;
END_IF
IF NOT(InitZeros(Size,Size)) THEN
	InitMagicSquare := FALSE;
	RETURN;
END_IF

InitMagicSquare := TRUE;

Ri := (Rows - 1)/2;
Ci := Cols-1;

FOR I := 1 TO Length DO
	SetRC(Ri,Ci,I);
	IF GetRC((Ri + 1) MOD Rows,(Ci + 1) MOD Cols) = 0 THEN
		Ri := (Ri + 1) MOD Rows;
		Ci := (Ci + 1) MOD Cols;
	ELSE
		IF Ci = 0 THEN
			Ci := Cols-1;
		ELSE
			Ci := Ci - 1;
		END_IF
	END_IF
END_FOR
END_METHOD

METHOD PUBLIC InitTrapezoidal : BOOL
VAR_INPUT
	Rows : UINT;
	Cols : UINT;
	Diagonal : LREAL;
	UpperRight : LREAL;
	LowerLeft : LREAL;
END_VAR
IF NOT(Init(Rows,Cols)) THEN
	InitTrapezoidal := FALSE;
	RETURN;
END_IF

InitTrapezoidal := TRUE;

FillTrapezoidal(Diagonal,UpperRight,LowerLeft);
END_METHOD

METHOD PUBLIC InitVector : BOOL
VAR_INPUT
	Length : UINT;
	Value : LREAL;
	Increment : LREAL;
END_VAR
IF NOT(Init(Length,1)) THEN
	InitVector := FALSE;
	RETURN;
END_IF

InitVector := TRUE;

IF Increment = 0 THEN
	FillTrapezoidal(Value,Value,Value);
ELSE
	IF Length > 0 THEN
		FOR I:= 0 TO Length-1 DO
			SetI(I,Value + I * Increment);
		END_FOR
	END_IF;
END_IF
END_METHOD

METHOD PUBLIC InitZeros : BOOL
VAR_INPUT
	Rows : UINT;
	Cols : UINT;
END_VAR
InitZeros := Resize(Rows,Cols,FALSE,TRUE);
END_METHOD

METHOD PUBLIC Grow : BOOL
VAR_INPUT
	Row : UINT;
	Col : UINT;
	DiagVal : LREAL;
	RowVal : LREAL;
	ColVal : LREAL;
END_VAR
VAR
	Temp : DynamicMatrix;
END_VAR
Temp.InitCopy(THIS^);
Grow := AsGrown(Temp,Row,Col,DiagVal,RowVal,ColVal);
END_METHOD

METHOD PUBLIC Resize : BOOL
VAR_INPUT
	NewRows : UINT;
	NewCols : UINT;
	RetainVals : BOOL;//retains 
	ClearVals : BOOL;
END_VAR
VAR
	OldData : POINTER TO LREAL;
	OldRows : UINT;
	OldCols : UINT;
END_VAR
//case where desired size is an empty matrix
IF NewRows * NewCols = 0 THEN
	IF Data <> 0 THEN
		MemManager.Free2(Data);
	END_IF
	
	Resize := TRUE;
	Rows_ := NewRows;
	Cols_ := NewCols;
	
//case where desired size is a non=empty matrix
ELSE
	//backup data so we can refill with it if necessary, then free it
	OldData := Data;
	OldRows := Rows;
	OldCols := Cols;
	
	//change primary buffer size
	Data := MemManager.Alloc(nSize := UINT_TO_UDINT(NewRows) * UINT_TO_UDINT(NewCols) * SIZEOF(LREAL), bReset := ClearVals);
	//error condition if memory cannot be allocated
	IF Data = 0 THEN
		Rows_ := 0;
		Cols_ := 0;
		ADSLOGSTR(ADSLOG_MSGTYPE_ERROR,'Unable to allocate memory when resizing matrix','');
		Resize := FALSE;
		Data := OldData;//put the data back, if any
		RETURN;
	END_IF
	
	Rows_ := NewRows;
	Cols_ := newCols;
	Resize := TRUE;
	
	//copy data if the previous size was not empty, the pointer is not null, and retain was selected
	IF RetainVals THEN
		IF NOT(OldRows*OldCols = 0) AND OldData <> 0 THEN
			FOR Ri := 0 TO MIN(NewRows,OldRows)-1 DO
				FOR Ci := 0 TO MIN(NewCols,OldCOls)-1 DO
					Data[RCC2I(Ri,Ci,NewCols)] := OldData[RCC2I(Ri,Ci,OldCols)];
				END_FOR
			END_FOR
		ELSE
			LogWarning('%s: Data retention optino was selected for resize, but the previous matrix did not have any data stored');
		END_IF
	END_IF
	
	//free old data now that everything works
	IF OldData <> 0 THEN
		MemManager.Free2(OldData);
	END_IF
	
	
	
END_IF
END_METHOD

METHOD PUBLIC Shrink : BOOL
VAR_INPUT
	Row : UINT;
	Col : UINT;
END_VAR
VAR
	Temp : DynamicMatrix;
END_VAR
IF IsEmpty THEN
	Shrink := FALSE;
	RETURN;
END_IF

Temp.InitCopy(THIS^);
Shrink := AsShrunk(Temp,Row,Col);
END_METHOD

METHOD PUBLIC Transpose : BOOL
VAR_INPUT
END_VAR
VAR
	Temp : DynamicMatrix;
END_VAR
IF IsSquare THEN
	Matrix_TransposeSquare(THIS^);
	Transpose := TRUE;
ELSE

	IF NOT(Temp.InitCopy(THIS^)) THEN
		Transpose := FALSE;
	END_IF
	
	Transpose := AsTransposed(Temp);

END_IF
END_METHOD

//Total number of columns in this matrix
PROPERTY PUBLIC Cols : UINT
GET
Cols := Cols_;
END_GET
END_PROPERTY

METHOD FB_exit : BOOL
VAR_INPUT
	bInCopyCode : BOOL; // if TRUE, the exit method is called for exiting an instance that is copied afterwards (online change).
END_VAR
IF NOT(bInCopyCode)THEN
	Free();
END_IF
END_METHOD

METHOD FB_init : BOOL
VAR_INPUT
	bInitRetains : BOOL; // if TRUE, the retain variables are initialized (warm start / cold start)
	bInCopyCode : BOOL;  // if TRUE, the instance afterwards gets moved into the copy code (online change)
END_VAR
Free();
END_METHOD

//Gets the value of the element in this matrix at the supplied location as if the elements were stored in a 1D row-major array
//:Prerequisites:
// - I < Rows*Cols
// - Matrix is not empty
//If the supplied index is out of bounds the value 0 is returned and a warning is generated in the Error List
METHOD PUBLIC GetI : LREAL//The value of the element at the specified index, or 0 if an invalid index is supplied
VAR_INPUT
	I : UINT;//The index of the element which should have its value returned
END_VAR
IF Data = 0 THEN
	GetI := 0.0;
	LogWarning('%s: Attempted I access of uninitialized Matrix');
ELSIF I >= Length THEN
	GetI := 0.0;
	LogWarning('%s: Attempted I access of out-of-bounds Matrix data');
ELSE
	GetI := Data[I];
END_IF
END_METHOD

//Total number of rows in this matrix
PROPERTY PUBLIC Rows : UINT
GET
Rows := Rows_;
END_GET
END_PROPERTY

//Sets the element specified by the supplied index to the suppleid value, assuming the data of the matrix is stored in a 1D row-major array
//:Prerequisites: - I < Rows*Cols
METHOD PUBLIC SetI : BOOL//TRUE if the specified index is valid and the data is copied. FLASE otherwise
VAR_INPUT
	I : UINT;//The index specifying which element should be modified
	Val : LREAL;//The value copied to the corresponding element
END_VAR
IF Data = 0 THEN
	SetI := FALSE;
	LogWarning('%s: Attempt to set data using I access when data is not initialized');
ELSIF I >= Length THEN
	SetI := FALSE;
	LogWarning('%s: Attempt to set data using I access when I is out of bounds');
ELSE
	SetI := TRUE;
	Data[I] := Val;
END_IF
END_METHOD

//Resets the content of this matrix to be a column vector, copied from the specified column of the input matrix
METHOD PUBLIC AsColVector : BOOL
VAR_IN_OUT CONSTANT
	M : Matrix;
END_VAR
VAR_INPUT
	Col : UINT;
END_VAR
AsColVector := AsSubMatrix(
	M := M,
	RowStart := 0,
	RowCount := M.Rows,
	ColStart := Col,
	ColCount := 1);
END_METHOD

//resets the content of this matrix to be the result of subtracting the input subtrahend matrix from the input minuend matrix element by element
METHOD PUBLIC AsElementDifference : BOOL
VAR_IN_OUT CONSTANT
	Minuend : Matrix;
	Subtrahend : Matrix;
END_VAR
IF NOT(Minuend.IsEqualSize(subtrahend)) THEN
	AsElementDifference := FALSE;
	LogWarning('%s: Matricies supplied to AsElementDifference were not the same size');
	RETURN;
END_IF

IF NOT(Init(Minuend.Rows,Minuend.Cols)) THEN
	AsElementDifference := FALSE;
	RETURN;
END_IF

AsElementDifference := Matrix_ElementSum(Minuend,Subtrahend,THIS^);
END_METHOD

//resets the content of this matrix to be the result of multiplying the input matricies element by element
METHOD PUBLIC AsElementProduct : BOOL
VAR_IN_OUT CONSTANT
	A : Matrix;
	B : Matrix;
END_VAR
IF NOT(A.IsEqualSize(B)) THEN
	AsElementProduct := FALSE;
	LogWarning('%s: Matricies supplied to AsElementProduct were not the same size');
	RETURN;
END_IF

IF NOT(Init(A.Rows,A.Cols)) THEN
	AsElementProduct := FALSE;
	RETURN;
END_IF

AsElementProduct := Matrix_ElementProduct(A,B,THIS^);
END_METHOD

//resets the content of this matrix to be the result of adding the input matricies element by element
METHOD PUBLIC AsElementSum : BOOL
VAR_IN_OUT CONSTANT
	A : Matrix;
	B : Matrix;
END_VAR
IF NOT(A.IsEqualSize(B)) THEN
	AsElementSum := FALSE;
	LogWarning('%s: Matricies supplied to AsElementSum were not the same size');
	RETURN;
END_IF

IF NOT(Init(A.Rows,A.Cols)) THEN
	AsElementSum := FALSE;
	RETURN;
END_IF

AsElementSum := Matrix_ElementSum(A,B,THIS^);
END_METHOD

//resets the content of this matrix to be a larger (by one row and one column) matrix copy of the input matrix. Initial values of the new row, column, and diagonal are controlled by other inputs.
METHOD PUBLIC AsGrown : BOOL
VAR_IN_OUT CONSTANT
	M : Matrix;
END_VAR
VAR_INPUT
	Row : UINT;
	Col : UINT;
	DiagVal : LREAL;
	RowVal : LREAL;
	ColVal : LREAL;
END_VAR
IF NOT(Init(M.Rows+1,M.Cols+1)) THEN
	AsGrown := FALSE;
	LogWarning('%s: Matrix supplied to AsGrown was not the right size');
	RETURN;
END_IF

AsGrown := Matrix_Grow(M,THIS^,Row,Col,DiagVal,RowVal,ColVal);
END_METHOD

//resets the contents of this matrix to be the inverse of the input matrix.
METHOD PUBLIC AsInverse : BOOL
VAR_IN_OUT CONSTANT
	M : Matrix;
END_VAR
VAR_INPUT
	//Values with a lower magnitude than the tolerance will be rounded to zero in order to avoid divide-by-near-zero situations
	Tolerance : LREAL;
END_VAR
IF NOT(M.IsSquare) OR M.IsEmpty THEN
	AsInverse := FALSE;
	RETURN;
END_IF

THIS^.InitCopy(M);
AsInverse := THIS^.InvertSquare(Tolerance);
END_METHOD

//resets the content of this matrix to be the product of input matrix A x input matrix B
METHOD PUBLIC AsMatrixProduct : BOOL
VAR_IN_OUT CONSTANT
	A : Matrix;
	B : Matrix;
END_VAR
IF A.Cols <> B.Rows THEN
	AsMatrixProduct := FALSE;
	LogWarning('%s: Matricies supplied to AsMatrixProduct are not compatible for multiplication');
	RETURN;
END_IF

IF NOT(Init(A.Rows,B.Cols)) THEN
	AsMatrixProduct := FALSE;
	RETURN;
END_IF

AsMatrixProduct := Matrix_Product(A,B,THIS^);
END_METHOD

//Resets the content of this matrix to be a row vector, copied from the specified row of the input matrix
METHOD PUBLIC AsRowVector : BOOL
VAR_IN_OUT CONSTANT
	M : Matrix;
END_VAR

VAR_INPUT
	Row : UINT;
END_VAR
AsRowVector := AsSubMatrix(
	M := M,
	RowStart := Row,
	RowCount := 1,
	ColStart := 0,
	ColCount := M.Cols);
END_METHOD

//resets the contents of this matrix to be an element by element product of the input matrix and the input scalar
METHOD PUBLIC AsScaled : BOOL
VAR_IN_OUT CONSTANT
	M : Matrix;
END_VAR
VAR_INPUT
	Scalar : LREAL;
END_VAR
IF NOT(InitCopy(M)) THEN
	AsScaled := FALSE;
	RETURN;
END_IF

AsScaled := TRUE;
Scale(Scalar);
END_METHOD

//resets the contents of this matrix to be a copy of the input matrix with one fewer row and column (the specified row and column are removed)
METHOD PUBLIC AsShrunk : BOOL
VAR_IN_OUT CONSTANT
	M : Matrix;
END_VAR
VAR_INPUT
	Row : UINT;
	Col : UINT;
END_VAR
IF NOT(Init(M.Rows-1,M.Cols-1)) THEN
	AsShrunk := FALSE;
	LogWarning('%s: Matrix supplied to AsGrown was not the right size');
	RETURN;
END_IF

AsShrunk := Matrix_Shrink(M,THIS^,Row,Col);
END_METHOD

//resets the contents of this matrix to be a copy of a continuous submatrix of the input reference matrix
METHOD PUBLIC AsSubMatrix : BOOL
VAR_IN_OUT CONSTANT
	M : Matrix;
END_VAR
VAR_INPUT
	RowStart : UINT;
	RowCount : UINT;
	ColStart : UINT;
	ColCount : UINT;
END_VAR
IF RowStart + RowCount > M.Rows THEN
	AsSubMatrix := FALSE;
	LogWarning('%s: Attempt to access out of bounds Row during SubMatrix access');
	RETURN;
END_IF
IF ColStart + ColCount > M.Cols THEN
	AsSubMatrix := FALSE;
	LogWarning('%s: Attempt to access out of bounds Row during SubMatrix access');
	RETURN;
END_IF

IF NOT(Init(RowCount,ColCount)) THEN
	AsSubMatrix := FALSE;
	RETURN;
END_IF

AsSubMatrix := Matrix_SubMatrix(M,THIS^,RowStart,RowCount,ColStart,ColCount);
END_METHOD

//Resets the contents of this matrix to be a transposed copy of the input matrix
METHOD PUBLIC AsTransposed : BOOL
VAR_IN_OUT CONSTANT
	M : Matrix;
END_VAR
IF NOT(Init(M.Cols,M.Rows)) THEN
	AsTransposed := FALSE;
	RETURN;
END_IF

AsTransposed := Matrix_Transpose(M,THIS^);
END_METHOD

//resets the contents of this matrix to be the result of a sequential vector cross product of all of the input matricies
METHOD PUBLIC AsVectorCrossProduct : BOOL
VAR_INPUT
END_VAR
VAR_IN_OUT CONSTANT
	Vectors : ARRAY[*] OF POINTER TO Matrix;
END_VAR
VAR
	Dim : UINT;
	Vi : DINT;
END_VAR
Dim := DINT_TO_UINT(UPPER_BOUND(Vectors,1) - LOWER_BOUND(Vectors,1))+2;

FOR I := 0 TO Dim-2 DO
	Vi := LOWER_BOUND(Vectors,1)+I;
	//check pointer before other checks because PLCs don't do short-circuit logic
	IF Vectors[Vi] = 0 THEN
		AsVectorCrossProduct := FALSE;
		LogWarning('%s: At least one of the elements of the Vector array is a null pointer');
		RETURN;
	END_IF
	IF Vectors[Vi]^.IsEmpty OR NOT(Vectors[Vi]^.IsVector) OR Vectors[Vi]^.Length <> Dim THEN
		AsVectorCrossProduct := FALSE;
		LogWarning('%s: At least one of the elements of the Vector array is empty, or not a vector of the right size');
		RETURN;
	END_IF
END_FOR

//only allocate memory if we think it will work
IF NOT(Init(Dim,1)) THEN
	AsVectorCrossProduct := FALSE;
	RETURN;
END_IF

AsVectorCrossProduct := Vector_CrossProduct(Res := THIS^, Vectors := Vectors);
END_METHOD

END_FUNCTION_BLOCK

// POUs/Functions/Arrays/Array2D_To_Matrix
FUNCTION Array2D_To_Matrix : BOOL
VAR_IN_OUT CONSTANT
	A : ARRAY[*,*] OF LREAL;//source matrix for element copy operation
END_VAR
VAR_IN_OUT
	M : Matrix;//destination matrix for element copy operation
END_VAR
VAR
	Ri : UINT;
	Ci : UINT;
	R0 : UINT;
	C0 : UINT;
END_VAR

//check for bad references and size agreement
IF NOT(Matrix_SameSizeAs_Array2D(A,M)) THEN
	Array2D_To_Matrix := FALSE;
	RETURN;
END_IF
Array2D_To_Matrix := TRUE;

R0 := DINT_TO_UINT(LOWER_BOUND(A,1));
C0 := DINT_TO_UINT(LOWER_BOUND(A,2));

IF M.IsEmpty THEN
	RETURN;//do not start loop when empty
END_IF

FOR Ri := 0 TO M.Rows-1 DO
	FOR Ci := 0 TO M.Cols-1 DO
		M.SetRC(Ri,Ci,A[R0+Ri,C0+Ci]);
	END_FOR
END_FOR

END_FUNCTION

// POUs/Functions/Arrays/Matrix_SameSizeAs_Array2D
FUNCTION Matrix_SameSizeAs_Array2D : BOOL
VAR_IN_OUT CONSTANT
	A : ARRAY[*,*] OF LREAL;
	M : Matrix;
END_VAR

//check for size mismatch
Matrix_SameSizeAs_Array2D := Array2D_Rows(A) = M.Rows AND Array2D_Cols(A) = M.Cols;

END_FUNCTION

// POUs/Functions/Arrays/Array2D_Rows
FUNCTION Array2D_Rows : UINT
VAR_IN_OUT CONSTANT
	A : ARRAY[*,*] OF LREAL;
END_VAR

IF UPPER_BOUND(A,1) < LOWER_BOUND(A,1) THEN
	Array2D_Rows := 0;
ELSE
	Array2D_Rows := DINT_TO_UINT(UPPER_BOUND(A,1) - LOWER_BOUND(A,1) + 1);
END_IF

END_FUNCTION

// POUs/Functions/Arrays/Array2D_Cols
FUNCTION Array2D_Cols : UINT
VAR_IN_OUT CONSTANT
	A : ARRAY[*,*] OF LREAL;
END_VAR

IF UPPER_BOUND(A,2) < LOWER_BOUND(A,2) THEN
	Array2D_Cols := 0;
ELSE
	Array2D_Cols := DINT_TO_UINT(UPPER_BOUND(A,2) - LOWER_BOUND(A,2) + 1);
END_IF

END_FUNCTION

// POUs/Functions/Matrix/Matrix_TransposeSquare
FUNCTION Matrix_TransposeSquare : BOOL
VAR_IN_OUT
	M : Matrix;
END_VAR
VAR
	Ri : UINT;
	Ci : UINT;
	Temp : LREAL;
END_VAR

IF NOT(M.IsSquare) OR M.isempty THEN
	Matrix_TransposeSquare := FALSE;
	RETURN;
END_IF

Matrix_TransposeSquare := TRUE;

IF M.Length <= 1 THEN
	RETURN;
END_IF

FOR Ri := 0 TO M.Rows-2 DO
	FOR Ci := Ri+1 TO M.Cols-1 DO
		M.SwapRC(Ri,Ci,Ci,Ri);
	END_FOR
END_FOR

END_FUNCTION

// POUs/Functions/Matrix/Matrix_ElementSum
FUNCTION Matrix_ElementSum : BOOL
VAR_IN_OUT CONSTANT
	A : Matrix;
	B : Matrix;
END_VAR
VAR_IN_OUT
	Res : Matrix;
END_VAR
VAR
	I : UINT;
END_VAR

IF NOT(A.IsEqualSize(Res)) OR A.IsEmpty THEN
	Matrix_ElementSum := FALSE;
	RETURN;
END_IF

IF NOT(B.IsEqualSize(Res)) OR B.IsEmpty THEN
	Matrix_ElementSum := FALSE;
	RETURN;
END_IF

Matrix_ElementSum := TRUE;

FOR I := 0 TO Res.Length - 1 DO
	Res.SetI(I,A.GetI(I)+B.GetI(I));
END_FOR

END_FUNCTION

// POUs/Functions/Matrix/Matrix_ElementProduct
FUNCTION Matrix_ElementProduct : BOOL
VAR_IN_OUT CONSTANT
	A : Matrix;
	B : Matrix;
END_VAR
VAR_IN_OUT
	Res : Matrix;
END_VAR
VAR
	I : UINT;
END_VAR

IF NOT(A.IsEqualSize(Res)) OR A.IsEmpty THEN
	Matrix_ElementProduct := FALSE;
	RETURN;
END_IF

IF NOT(B.IsEqualSize(Res)) OR B.IsEmpty THEN
	Matrix_ElementProduct := FALSE;
	RETURN;
END_IF

Matrix_ElementProduct := TRUE;

FOR I := 0 TO Res.Length - 1 DO
	Res.SetI(I,A.GetI(I)*B.GetI(I));
END_FOR

END_FUNCTION

// POUs/Functions/Matrix/Matrix_Grow
FUNCTION Matrix_Grow : Bool
VAR_IN_OUT CONSTANT
	M_From : Matrix;
END_VAR
VAR_IN_OUT
	M_To : Matrix;
END_VAR
VAR_INPUT
	Row : UINT;
	Col : UINT;
	DiagVal : LREAL;
	RowVal : LREAL;
	ColVal : LREAL;
END_VAR


VAR
	Ri : UINT;
	Ci : UINT;
END_VAR

IF M_From.Rows <> M_To.Rows-1 THEN
	Matrix_Grow := FALSE;
	RETURN;
END_IF
IF M_From.Cols <> M_To.Cols-1 THEN
	Matrix_Grow := FALSE;
	RETURN;
END_IF

IF Row < 0 OR Row > M_From.Rows THEN
	Matrix_Grow := FALSE;
	RETURN;
END_IF

IF Col < 0 OR Col > M_From.Cols THEN
	Matrix_Grow := FALSE;
	RETURN;
END_IF

Matrix_Grow := TRUE;

//loop backwards to avoid possible overwriting the input if the same matrix is both inputs.
//in order to ensure the final decrement breaks the loop condition the final valid value must be 1, not zero. So just offset all indexes by 1...
FOR Ri := 0 TO M_To.Rows-1 DO
	FOR Ci := 0 TO M_To.Cols-1 DO
		IF Ri = Row AND Ci = Col THEN
			M_To.SetRC(Ri,Ci,DiagVal);
		ELSIF Ri = Row THEN
			M_To.SetRC(Ri,Ci,RowVal);
		ELSIF Ci = Col THEN
			M_To.SetRC(Ri,Ci,ColVal);
		ELSE
			//note that if Ri or Ci is their lowest value (1), then the BOOL condition must be false because 0 cannot be greater than any UINT.
			//This guarantees that the lowest RC indexes are zero.
			M_To.SetRC(Ri,Ci,M_From.GetRC(Ri - BOOL_TO_UINT((Ri)>Row),Ci - BOOL_TO_UINT((Ci)>Col)));
		END_IF
	END_FOR
END_FOR

END_FUNCTION

// POUs/Functions/Matrix/Matrix_Product
FUNCTION Matrix_Product : Bool
VAR_IN_OUT CONSTANT
	A : Matrix;//left side matrix
	B : Matrix;//right side matrix
END_VAR
VAR_IN_OUT
	Res : Matrix;//must not be the same source as M_L or M_R
END_VAR
VAR
	Ri : UINT;
	Ci : UINT;
	I : UINT;
	Sum : LREAL;
END_VAR

IF NOT(Matrix_CanMult(A,B)) THEN
	Matrix_Product := FALSE;
	RETURN;
END_IF

IF A.Rows <> Res.Rows OR B.Cols <> Res.Cols THEN
	Matrix_Product := FALSE;
	RETURN;
END_IF

Matrix_Product := TRUE;

FOR Ri := 0 TO Res.Rows-1 DO
	FOR Ci := 0 TO Res.Cols-1 DO
		Sum := 0;
		FOR I := 0 TO A.Cols-1 DO
			Sum := Sum + A.GetRC(Ri,I) * B.GetRC(I,Ci);
		END_FOR
		Res.SetRC(Ri,Ci,Sum);
	END_FOR
END_FOR

END_FUNCTION

// POUs/Functions/Matrix/Matrix_CanMult
FUNCTION Matrix_CanMult : Bool
VAR_IN_OUT CONSTANT
	M_L : Matrix;
	M_R : Matrix;
END_VAR
VAR
END_VAR

Matrix_CanMult := NOT(M_L.IsEmpty) AND NOT(M_R.IsEmpty) AND M_L.Cols = M_R.Rows;

END_FUNCTION

// POUs/Functions/Matrix/Matrix_Shrink
FUNCTION Matrix_Shrink : Bool
VAR_IN_OUT CONSTANT
	M_From : Matrix;
END_VAR
VAR_IN_OUT
	M_To : Matrix;
END_VAR
VAR_INPUT
	Row : UINT;
	Col : UINT;
END_VAR


VAR
	Ri : UINT;
	Ci : UINT;
END_VAR

IF M_From.Length <= 1 THEN
	Matrix_Shrink := FALSE;
	RETURN;
END_IF

IF M_To.Rows <> MAX(1,M_From.Rows-1) OR M_To.Cols <> MAX(1,M_From.Cols-1) THEN
	Matrix_Shrink := FALSE;
	RETURN;
END_IF

IF Row >= M_From.Rows OR Col >= M_From.Cols THEN
	Matrix_Shrink := FALSE;
	RETURN;
END_IF

Matrix_Shrink := TRUE;

FOR Ri := 0 TO M_To.Rows-1 DO
	FOR Ci := 0 TO M_To.Cols-1 DO
		M_To.SetRC(Ri,Ci,M_From.GetRC(Ri + BOOL_TO_UINT(Ri >= Row AND M_From.Rows <> M_To.Rows),Ci + BOOL_TO_UINT(Ci >= Col AND M_From.Cols <> M_To.Cols)));
	END_FOR
END_FOR

END_FUNCTION

// POUs/Functions/Matrix/Matrix_SubMatrix
FUNCTION Matrix_SubMatrix : Bool
VAR_IN_OUT CONSTANT
	M_Super : Matrix;
END_VAR
VAR_IN_OUT
	M_Sub : Matrix;
END_VAR
VAR_INPUT
	RowStart : UINT;
	RowCount : UINT;
	ColStart : UINT;
	ColCount : UINT;
END_VAR


VAR
	Ri : UINT;
	Ci : UINT;
END_VAR

IF RowStart + RowCount > M_Super.Rows OR ColStart + ColCount > M_Super.Cols THEN
	Matrix_SubMatrix := FALSE;
	RETURN;
END_IF
IF M_Sub.Rows <> RowCount  OR M_Sub.Cols <> ColCount THEN
	Matrix_SubMatrix := FALSE;
	RETURN;
END_IF

Matrix_SubMatrix := TRUE;

IF RowCount = 0 OR ColCount = 0 THEN
	RETURN;//valid to get a zero-len matrix as the result, but indexing below will cause a pagefault due to creating 32k+ warning messages for invalid access
END_IF

FOR Ri := 0 TO RowCount-1 DO
	FOR Ci := 0 TO ColCount-1 DO
		M_Sub.SetRC(Ri,Ci,M_Super.GetRC(RowStart+Ri,ColStart+Ci));
	END_FOR
END_FOR

END_FUNCTION

// POUs/Functions/Matrix/Matrix_Transpose
FUNCTION Matrix_Transpose : Bool
VAR_IN_OUT CONSTANT
	M_From : Matrix;
END_VAR
VAR_IN_OUT
	M_To : Matrix;
END_VAR
VAR
	Ri : UINT;
	Ci : UINT;
END_VAR

IF M_From.Rows <> M_To.Cols OR M_From.Cols <> M_to.Rows THEN
	Matrix_Transpose := FALSE;
	RETURN;
END_IF

Matrix_Transpose := TRUE;

FOR Ri := 0 TO M_From.Rows-1 DO
	FOR Ci := 0 TO M_From.Cols-1 DO
		M_To.SetRC(Ci,Ri,M_From.GetRC(Ri,Ci));
	END_FOR
END_FOR

END_FUNCTION

// POUs/Functions/Vector/Vector_CrossProduct
FUNCTION Vector_CrossProduct : BOOL
VAR_IN_OUT
	Res : Matrix;
END_VAR
VAR_IN_OUT CONSTANT
	Vectors : ARRAY[*] OF POINTER TO Matrix;
END_VAR
VAR
	Ri : UINT;
	Ci : UINT;
	I : DINT;
	M_Vectors : DynamicMatrix;
	M_Det : ShrunkMatrixAccessor;
	Det : LREAL;
	Sign : LREAL;
END_VAR

//a cross product in N dimensions space requires N-1 vectors of length N, the result of which is an N-length vector orthogonal to all supplied vectors. Order of vectors matters.
//if you arrange all supplied vectors horizontally into an almost-square matrix, then each component of the result vector is simply the determinate of the aggregate matrix with the corresponding column removed

IF NOT(Res.IsVector) OR Res.IsEmpty OR (UPPER_BOUND(Vectors,1) - LOWER_BOUND(Vectors,1) + 1) <> Res.Length - 1 THEN
	Vector_CrossProduct := FALSE;
	RETURN;
END_IF

FOR I := LOWER_BOUND(Vectors,1) TO UPPER_BOUND(Vectors,1) DO
	IF Vectors[I] = 0 THEN
		Vector_CrossProduct := FALSE;
		RETURN;
	END_IF
	IF NOT(Vectors[I]^.IsVector) OR Vectors[I]^.Length <> Res.Length THEN
		Vector_CrossProduct := FALSE;
		RETURN;
	END_IF
END_FOR


IF NOT(M_Vectors.Init(Res.Length,Res.Length)) THEN
	Vector_CrossProduct := FALSE;
	RETURN;
END_IF


//build aggregate matrix
FOR Ri := 0 TO M_Vectors.Rows-1 DO
	FOR Ci := 0 TO M_Vectors.Cols-1 DO
		IF Ri = 0 THEN
			M_Vectors.SetRC(Ri,Ci,1);
		ELSE
			I := LOWER_BOUND(Vectors,1)-1 + Ri;
			M_Vectors.SetRC(Ri,Ci,Vectors[I]^.GetI(Ci));
		END_IF
	END_FOR
END_FOR

//if some vectors are parallel or whatever there is no 'one' cross product, so return false
IF M_Vectors.GetDeterminant() = 0 THEN
	Vector_CrossProduct := FALSE;
	RETURN;
END_IF

Vector_CrossProduct := TRUE;

//take determiantes
FOR Ci := 0 TO M_Vectors.Cols-1 DO
	M_Det.Init(M_Vectors,0,Ci);
	IF NOT(Matrix_DeterminateSquare(M_Det, Res=>Det)) THEN
		Vector_CrossProduct := FALSE;
		RETURN;
	END_IF
	Sign := ((UINT_TO_INT(Ci)+1) MOD 2)*2 -1;//even columns are positive, odd columns are negative
	Res.SetI(Ci,Det*Sign);
END_FOR

END_FUNCTION

// POUs/Functions/Matrix/Matrix_DeterminateSquare
FUNCTION Matrix_DeterminateSquare : BOOL
VAR_IN_OUT CONSTANT
	M : Matrix;
END_VAR
VAR_OUTPUT
	Res : LREAL;
END_VAR
VAR
	Sum : LREAL;
	Sign : LREAL;
	SubMatrix : ShrunkMatrixAccessor;
	
	Ci : UINT;
END_VAR

IF NOT(M.IsSquare) OR M.IsEmpty THEN
	Matrix_DeterminateSquare := FALSE;
	Res := 0;
	RETURN;
END_IF

Matrix_DeterminateSquare := TRUE;

IF M.Length = 1 THEN
	Res := M.GetRC(0,0);
ELSE
	Sum := 0;
	FOR Ci := 0 TO M.Cols-1 DO
		Sign := ((UINT_TO_INT(Ci)+1) MOD 2)*2 -1;//even columns are positive, odd columns are negative
		SubMatrix := M.GetShrunkMatrixAccessor(0,Ci);
		Sum := Sum + Sign * M.GetRC(0,Ci) * SubMatrix.GetDeterminant();//direct recursion is not accessible, but this should work
	END_FOR
	Res := Sum;
END_IF

END_FUNCTION

// POUs/MatrixAccessors/ShrunkMatrixAccessor
FUNCTION_BLOCK ShrunkMatrixAccessor EXTENDS MatrixAccessor
VAR_INPUT
END_VAR
VAR_OUTPUT
END_VAR
VAR
	RowRemoved_ : UINT;
	ColRemoved_ : UINT;
END_VAR

METHOD PUBLIC Init
VAR_INPUT
	M : REFERENCE TO Matrix;
	RowRemoved : UINT;
	ColRemoved : UINT;
END_VAR
Init_(M);
RowRemoved_ := RowRemoved;
ColRemoved_ := ColRemoved;
END_METHOD

//Total number of columns in this matrix
PROPERTY PUBLIC Cols : UINT
GET
IF NOT __ISVALIDREF(M_) THEN
	Cols := 0;
	LogWarning('%s Attempted Cols access using uninitialized Matrix Accessor');
ELSIF M_.Cols > 0 THEN
	Cols := M_.Cols-1;
ELSE
	Cols := 0;
END_IF
END_GET
END_PROPERTY

//Total number of rows in this matrix
PROPERTY PUBLIC Rows : UINT
GET
IF NOT __ISVALIDREF(M_) THEN
	Rows := 0;
	LogWarning('%s Attempted Rows access using uninitialized Matrix Accessor');
ELSIF M_.Rows > 0 THEN
	Rows := M_.Rows-1;
ELSE
	Rows := 0;
END_IF
END_GET
END_PROPERTY

METHOD PROTECTED This2Parent : UINT
VAR_INPUT
	Index : UINT;
END_VAR
VAR
	ThisR : UINT;
	ThisC : UINT;
END_VAR
IF NOT __ISVALIDREF(M_) THEN
	LogWarning('%s Attempted This2Parent calculation using uninitialized Matrix Accessor');
	This2Parent := 0;
	RETURN;
END_IF

IC2RC(Index,Cols,Row => ThisR, Col => ThisC);

This2Parent := RCC2I(ThisR+BOOL_TO_UINT(RowRemoved_<=ThisR),ThisC+BOOL_TO_UINT(ColRemoved_<=ThisC),M_.Cols);
END_METHOD

END_FUNCTION_BLOCK

// POUs/MatrixAccessors/MatrixAccessor
FUNCTION_BLOCK ABSTRACT MatrixAccessor EXTENDS Matrix
VAR_INPUT
END_VAR
VAR_OUTPUT
END_VAR
VAR
	M_ : REFERENCE TO Matrix;
END_VAR

METHOD PROTECTED Init_
VAR_INPUT
	M : REFERENCE TO Matrix;
END_VAR
M_ REF= M;
END_METHOD

METHOD PROTECTED This2Parent : UINT
VAR_INPUT
	Index : UINT;
END_VAR
This2Parent := Index;
END_METHOD

//Gets the value of the element in this matrix at the supplied location as if the elements were stored in a 1D row-major array
//:Prerequisites:
// - I < Rows*Cols
// - Matrix is not empty
//If the supplied index is out of bounds the value 0 is returned and a warning is generated in the Error List
METHOD PUBLIC GetI : LREAL//The value of the element at the specified index, or 0 if an invalid index is supplied
VAR_INPUT
	I : UINT;//The index of the element which should have its value returned
END_VAR
VAR
END_VAR
IF NOT __ISVALIDREF(M_) THEN
	GetI := 0.0;
	LogWarning('%s Attempted I access to uninitialized Matrix Accessor');
ELSIF IsEmpty THEN
	GetI := 0.0;
	LogWarning('%s: Attempted I access of empty Matrix Accessor');
ELSIF I >= Length THEN
	GetI := 0.0;
	LogWarning('%s: Attempted I access beyond limits of Matrix Accessor');
ELSE
	GetI := M_.GetI(This2Parent(I));
END_IF
END_METHOD

//Sets the element specified by the supplied index to the suppleid value, assuming the data of the matrix is stored in a 1D row-major array
//:Prerequisites: - I < Rows*Cols
METHOD PUBLIC SetI : BOOL//TRUE if the specified index is valid and the data is copied. FLASE otherwise
VAR_INPUT
	I : UINT;//The index specifying which element should be modified
	Val : LREAL;//The value copied to the corresponding element
END_VAR
IF NOT __ISVALIDREF(M_) THEN
	SetI := FALSE;
	LogWarning('%s Attempted I access to uninitialized Matrix Accessor');
ELSIF IsEmpty THEN
	SetI := FALSE;
	LogWarning('%s: Attempted I access of empty Matrix Accessor');
ELSIF I >= Length THEN
	SetI := FALSE;
	LogWarning('%s: Attempted I access beyond limits of Matrix Accessor');
ELSE
	SetI := M_.SetI(This2Parent(I),Val);
END_IF
END_METHOD

END_FUNCTION_BLOCK

// POUs/StaticMatrix
(*
Derived class must:
- Declare a VAR array of LREAL named Data_
- Call Init_ in FB_init, pointing to the local arrays, with Rows and Cols such that Rows*Cols <= Length(Data_)
*)
{attribute 'reflection'}
{attribute 'no_assign'}
FUNCTION_BLOCK ABSTRACT StaticMatrix EXTENDS Matrix
VAR_INPUT
END_VAR
VAR_OUTPUT
END_VAR
VAR
	Rows_ : UINT := 0;
	Cols_ : UINT := 0;
END_VAR

METHOD PROTECTED Init_
VAR_INPUT
	RowCount : UINT;
	ColCount : UINT;
END_VAR
Rows_ := RowCount;
Cols_ := ColCount;
END_METHOD

//Total number of columns in this matrix
PROPERTY PUBLIC Cols : UINT
GET
Cols := Cols_;
END_GET
END_PROPERTY

//Total number of rows in this matrix
PROPERTY PUBLIC Rows : UINT
GET
Rows := Rows_;
END_GET
END_PROPERTY

END_FUNCTION_BLOCK

// POUs/MatrixAccessors/SubMatrixAccessor
FUNCTION_BLOCK SubMatrixAccessor EXTENDS MatrixAccessor
VAR_INPUT
END_VAR
VAR_OUTPUT
END_VAR
VAR
	RowStart_ : UINT;
	RowCount_ : UINT;
	ColStart_ : UINT;
	ColCount_ : UINT;
END_VAR

METHOD PUBLIC Init
VAR_INPUT
	M : REFERENCE TO Matrix;
	RowStart : UINT;
	RowCount : UINT;
	ColStart : UINT;
	ColCount : UINT;
END_VAR
Init_(M);
RowStart_ := RowStart;
RowCount_ := RowCount;
ColStart_ := ColStart;
ColCount_ := ColCount;
END_METHOD

//Total number of columns in this matrix
PROPERTY PUBLIC Cols : UINT
GET
IF NOT __ISVALIDREF(M_) THEN
	Cols := 0;
	LogWarning('%s Attempted Cols access using uninitialized Matrix Accessor');
ELSIF ColStart_+ColCount_ > M_.Cols THEN
	Cols := 0;
ELSE
	Cols := ColCount_;
END_IF
END_GET
END_PROPERTY

//Total number of rows in this matrix
PROPERTY PUBLIC Rows : UINT
GET
IF NOT __ISVALIDREF(M_) THEN
	Rows := 0;
	LogWarning('%s Attempted Rows access using uninitialized Matrix Accessor');
ELSIF RowStart_+RowCount_ > M_.Rows THEN
	Rows := 0;
ELSE
	Rows := RowCount_;
END_IF
END_GET
END_PROPERTY

METHOD PROTECTED This2Parent : UINT
VAR_INPUT
	Index : UINT;
END_VAR
VAR
	ThisR : UINT;
	ThisC : UINT;
END_VAR
IF NOT __ISVALIDREF(M_) THEN
	LogWarning('%s Attempted This2Parent calculation using uninitialized Matrix Accessor');
	This2Parent := 0;
	RETURN;
END_IF

IC2RC(Index,Cols,Row => ThisR, Col => ThisC);
This2Parent := RCC2I(ThisR+RowStart_,ThisC+ColStart_,M_.Cols);
END_METHOD

END_FUNCTION_BLOCK

// POUs/MatrixAccessors/TransposeMatrixAccessor
FUNCTION_BLOCK TransposeMatrixAccessor EXTENDS MatrixAccessor
VAR_INPUT
END_VAR
VAR_OUTPUT
END_VAR
VAR
	RowRemoved_ : UINT;
	ColRemoved_ : UINT;
END_VAR

METHOD PUBLIC Init
VAR_INPUT
	M : REFERENCE TO Matrix;
END_VAR
Init_(M);
END_METHOD

//Total number of columns in this matrix
PROPERTY PUBLIC Cols : UINT
GET
IF NOT __ISVALIDREF(M_) THEN
	Cols := 0;
	LogWarning('%s Attempted Cols access using uninitialized Matrix Accessor');
ELSE
	Cols := M_.Rows;
END_IF
END_GET
END_PROPERTY

//Total number of rows in this matrix
PROPERTY PUBLIC Rows : UINT
GET
IF NOT __ISVALIDREF(M_) THEN
	Rows := 0;
	LogWarning('%s Attempted Rows access using uninitialized Matrix Accessor');
ELSE
	Rows := M_.Cols;
END_IF
END_GET
END_PROPERTY

METHOD PROTECTED This2Parent : UINT
VAR_INPUT
	Index : UINT;
END_VAR
VAR
	ThisR : UINT;
	ThisC : UINT;
END_VAR
IF NOT __ISVALIDREF(M_) THEN
	LogWarning('%s Attempted This2Parent calculation using uninitialized Matrix Accessor');
	This2Parent := 0;
	RETURN;
END_IF

IC2RC(Index,Cols,Row => ThisR, Col => ThisC);

This2Parent := RCC2I(ThisC,ThisR,M_.Cols);
END_METHOD

END_FUNCTION_BLOCK

// POUs/Functions/Vector/Vector_DotProduct
FUNCTION Vector_DotProduct : BOOL
VAR_IN_OUT CONSTANT
	A : Matrix;
	B : Matrix;
END_VAR
VAR_OUTPUT
	Res : LREAL;
END_VAR
VAR
	Sum : LREAL;
	I : UINT;
END_VAR

IF NOT(A.IsVector) OR NOT(B.IsVector) OR A.Length <> B.Length OR A.IsEmpty THEN
	Vector_DotProduct := FALSE;
	Res := 0;
	RETURN;
END_IF

Vector_DotProduct := TRUE;

Sum := 0;
FOR I := 0 TO A.Length-1 DO
	Sum := Sum + A.GetI(I)*B.GetI(I);
END_FOR
Res := SUM;

END_FUNCTION

// POUs/Functions/Vector/Vector_Magnitude
FUNCTION Vector_Magnitude : BOOL
VAR_IN_OUT CONSTANT
	IN : Matrix;
END_VAR
VAR_OUTPUT
	Res : LREAL;
END_VAR
VAR
	Sum : LREAL;
	I : UINT;
END_VAR

IF NOT(IN.IsVector) OR IN.IsEmpty THEN
	Res := 0;
	Vector_Magnitude := FALSE;
	RETURN;
END_IF

Vector_Magnitude := TRUE;
Sum := 0;

FOR I := 0 TO IN.Length-1 DO
	Sum := Sum + IN.GetI(I) * IN.GetI(I);
END_FOR

Res := SQRT(Sum);

END_FUNCTION

// POUs/Functions/Matrix/Matrix_Copy
FUNCTION Matrix_Copy : BOOL
VAR_IN_OUT CONSTANT
	M_From : Matrix;
END_VAR
VAR_IN_OUT
	M_To : Matrix;
END_VAR

IF M_From.IsEmpty OR M_To.IsEmpty OR NOT(M_From.IsEqualSize(M_To)) THEN
	Matrix_Copy := FALSE;
	RETURN;
END_IF

Matrix_Copy := TRUE;

M_To.FillFrom(M_From);

END_FUNCTION

// POUs/Functions/Matrix/Matrix_ElementDifference
//Res := Minuend - Subtrahend
FUNCTION Matrix_ElementDifference : BOOL
VAR_IN_OUT CONSTANT
	Minuend : Matrix;
	Subtrahend : Matrix;
END_VAR
VAR_IN_OUT
	Res : Matrix;
END_VAR
VAR
	I : UINT;
END_VAR

IF NOT(Minuend.IsEqualSize(Res)) OR Minuend.IsEmpty THEN
	Matrix_ElementDifference := FALSE;
	RETURN;
END_IF

IF NOT(Subtrahend.IsEqualSize(Res)) OR Subtrahend.IsEmpty THEN
	Matrix_ElementDifference := FALSE;
	RETURN;
END_IF

Matrix_ElementDifference := TRUE;

FOR I := 0 TO Res.Length - 1 DO
	Res.SetI(I,Minuend.GetI(I)-Subtrahend.GetI(I));
END_FOR

END_FUNCTION

// POUs/Functions/Matrix/Matrix_InvertSquare
FUNCTION Matrix_InvertSquare : BOOL
VAR_IN_OUT
	M : Matrix;
END_VAR
VAR_INPUT
	Tolerance : LREAL;//numbers with a smaller magnitude than this will not be used as denominators, sintead resulting in an abort
END_VAR

VAR
	Ri : UINT;
	Ci : UINT;
	Ni : UINT;
	Mi : UINT;
	temp : LREAL;
END_VAR

IF NOT(M.IsSquare)THEN
	Matrix_InvertSquare := FALSE;
	RETURN;
END_IF

Matrix_InvertSquare := TRUE;

IF M.Length <= 1 THEN
	RETURN;
END_IF

FOR Mi := 0 TO M.Cols-1 DO
	//for each element RC(Ni,Ni)....
	temp := M.GetRC(Mi,Mi);//used as denominator everywhere
	IF ABS(temp) < Tolerance THEN
		Matrix_InvertSquare := FALSE;
		RETURN;
	END_IF;
	
	//Kron reduction
	FOR Ri := 0 TO M.Rows-1 DO
		IF Ri <> Mi THEN
			FOR Ci := 0 TO M.Cols-1 DO
				IF Ci <> Mi THEN
					M.SetRC(Ri,Ci,M.GetRC(Ri,Ci) - M.GetRC(Ri,Mi)*M.GetRC(Mi,Ci)/temp);
				END_IF
			END_FOR
		END_IF;
	END_FOR
	
	temp := -1/temp;
	M.SetRC(Mi,Mi,temp);
	FOR Ni := 0 TO M.Cols-1 DO
		IF Ni <> Mi THEN
			M.SetRC(Mi,Ni,M.GetRC(Mi,Ni)*temp);
			M.SetRC(Ni,Mi,M.GetRC(Ni,Mi)*temp);
		END_IF;
	END_FOR
	
END_FOR

M.Scale(-1);

END_FUNCTION

// POUs/Functions/Matrix/Matrix_Scale
FUNCTION Matrix_Scale : BOOL
VAR_IN_OUT
	M : Matrix;
END_VAR
VAR_INPUT
	Scalar : LREAL;
END_VAR

VAR
	I : UINT;
END_VAR

Matrix_Scale := TRUE;

IF M.IsEmpty THEN
	RETURN;
END_IF

FOR I := 0 TO M.Length-1 DO
	M.SetI(I,Scalar * M.GetI(I));
END_FOR

END_FUNCTION

// POUs/Csv/MatrixCsvWriter
FUNCTION_BLOCK MatrixCsvWriter
VAR_IN_OUT
	M : Matrix;
END_VAR
VAR_INPUT
	bExecute : BOOL;
	sPathName : T_MaxString;
	tTimeout : TIME;//timeout applied indidivudally to each file operation
	pHeader : POINTER TO STRING;
	cbHeaderLen : UDINT;
END_VAR
VAR_OUTPUT
	bBusy : BOOL;
	bError : BOOL;
	nErrId : UDINT;
	nErrStep : UDINT;
END_VAR
VAR
	FileOpen : FB_FileOpen;
	CsvWrite : FB_CSVMemBufferWriter;
	FileWrite : FB_FileWrite;
	FileClose : FB_FileClose;
	
	hFile : UINT;
	buffer : STRING(bufferSize+1);
	bufferOffset : UINT;//0 or 1
	step : UDINT;
	
	Ri : UINT;
	Ci : UINT;
	BuffCmd : E_EnumCmdType;
END_VAR
VAR CONSTANT
	bufferSize : UDINT := 1024;
	dataSize : UDINT := 32;	

	stepReady : UDINT := 0;
	stepOpenFile : UDINT := 1;
	stepWriteHeader : UDINT := 2;
	stepFillBuffer : UDINT := 3;
	stepWriteBuffer : UDINT := 4;
	stepCloseFile : UDINT := 5;
	stepDone : UDINT := 6;
END_VAR

FileOpen(
			sNetId := '',
			sPathName := spathname,
			nMode := FOPEN_MODEWRITE OR FOPEN_MODEBINARY,
			ePath := E_OpenPath.PATH_GENERIC,
			bExecute := step = stepOpenFile,
			tTimeout := tTimeout);
FileWrite(snetId := '',
			hFile := hFile,
			//pWriteBuff := SET INDIVIDUALLY
			//cbWriteLen := SET INDIVIDUALLY
			bExecute := step = stepWriteBuffer OR step = stepWriteHeader,
			tTimeout := tTimeout);
FileClose(
			snetId := '',
			hFile := hFile,
			bexecute := step = stepCloseFile,
			tTimeout := tTimeout);
			
CASE step OF
	stepReady:
		bError := FALSE;
		nErrId := 0;
		nErrStep := 0;
		Ri := 0;
		Ci := 0;
		
		IF bExecute THEN
			IF NOT M.IsEmpty THEN
				bBusy := TRUE;
				step := stepOpenFile;
			END_IF
		END_IF
		
	stepOpenFile:
		
		IF FileOpen.bError THEN
			bError := TRUE;
			nErrId := FileOpen.nErrId;
			nErrStep := step;
			step := stepDone;
		ELSIF NOT(FileOpen.bBusy) THEN
			hFile := FileOpen.hFile;
			IF pHeader <> 0 AND cbHeaderLen > 0 THEN
				step := stepWriteHeader;
				FileWrite.pWriteBuff := pHeader;
				FileWrite.cbWriteLen := cbHeaderLen;
			ELSE
				step := stepFillBuffer;
			END_IF;
		END_IF
		
	stepWriteHeader:
		IF FileWrite.bError THEN
			bError := TRUE;
			nErrId := FileWrite.nErrId;
			nErrStep := step;
			step := stepCloseFile;
		ELSIF NOT(FileWrite.bBusy) THEN
			step := stepFillBuffer;
		END_IF
		
		
	stepFillBuffer:
		//add field divider manually at the beginning of the write block
		IF Ci > 0 THEN
			buffer[0] := DEFAULT_CSV_FIELD_SEP;
			bufferOffset := 1;
		ELSE
			bufferOffset := 0;
		END_IF
		
		BuffCmd := E_EnumCmdType.eEnumCmd_First;
		REPEAT
			CsvWrite(eCmd := BuffCmd,
				putValue := LREAL_TO_STRING(M.GetRC(Ri,Ci)),
				bCRLF := M.Cols = Ci+1,
				pBuffer := ADR(buffer)+bufferOffset,
				cbBuffer := bufferSize-bufferOffset);
				
			IF NOT(CsvWrite.bOk) THEN
				bError := TRUE;
				nErrId := 1;
				nErrStep := step;
				step := stepCloseFile;
				RETURN;
			END_IF
				
			BuffCmd := E_EnumCmdType.eEnumCmd_Next;
			Ci := Ci + 1;
			IF Ci >= M.Cols THEN
				Ci := 0;
				Ri := Ri + 1;
			END_IF
		UNTIL 
			Ri >= M.Rows OR CsvWrite.cbFree < dataSize
		END_REPEAT 
		step := stepWriteBuffer;
		FileWrite.pWriteBuff := ADR(buffer);
		FileWrite.cbWriteLen := CsvWrite.cbSize+bufferOffset;
		
		
	stepWriteBuffer:
		
		IF FileWrite.bError THEN
			bError := TRUE;
			nErrId := FileWrite.nErrId;
			nErrStep := step;
			step := stepDone;
		ELSIF NOT(FileWrite.bBusy) THEN
			IF Ri >= M.Rows THEN
				step := stepCloseFile;
			ELSE
				step := stepFillBuffer;
			END_IF
		END_IF
		
	stepCloseFile:
		
		IF FileClose.bError AND NOT bError THEN
			bError := TRUE;
			nErrId := FileClose.nErrId;
			nErrStep := step;
			step := stepDone;
		ELSIF NOT(FileClose.bBusy) THEN
			step := stepDone;
		END_IF
		
		
	stepDone:
		bBusy := FALSE;
END_CASE

IF NOT bExecute THEN
	step := stepReady;
	bBusy := FALSE;
END_IF

END_FUNCTION_BLOCK

// POUs/Functions/Arrays/Matrix_To_Array2D
FUNCTION Matrix_To_Array2D : BOOL
VAR_IN_OUT
	A : ARRAY[*,*] OF LREAL;//destination matrix for element copy operation
END_VAR
VAR_IN_OUT CONSTANT
	M : Matrix;//source matrix for element copy operation
END_VAR
VAR
	Ri : UINT;
	Ci : UINT;
	R0 : UINT;
	C0 : UINT;
END_VAR

//check for bad references and size agreement
IF NOT(Matrix_SameSizeAs_Array2D(A,M)) THEN
	Matrix_To_Array2D := FALSE;
	RETURN;
END_IF
Matrix_To_Array2D := TRUE;

R0 := DINT_TO_UINT(LOWER_BOUND(A,1));
C0 := DINT_TO_UINT(LOWER_BOUND(A,2));

IF M.IsEmpty THEN
	RETURN;//do not start loop when empty
END_IF

FOR Ri := 0 TO M.Rows-1 DO
	FOR Ci := 0 TO M.Cols-1 DO
		A[R0+Ri,C0+Ci] := M.GetRC(Ri,Ci);
	END_FOR
END_FOR

END_FUNCTION

// POUs/Functions/Vector/Vector_Normalize
FUNCTION Vector_Normalize : BOOL
VAR_IN_OUT CONSTANT
	In : Matrix;
END_VAR
VAR_IN_OUT
	Res : Matrix;
END_VAR
VAR
	Mag : LREAL;
	I : UINT;
END_VAR

IF NOT(IN.IsVector) OR NOT(Res.IsVector) OR IN.IsEmpty OR IN.Length <> Res.Length THEN
	Vector_Normalize := FALSE;
	RETURN;
END_IF

IF NOT(Vector_Magnitude(In,Res=>Mag)) THEN
	Vector_Normalize := FALSE;
	RETURN;
END_IF

//dont use copy because vectors might be in different orientations
FOR I:= 0 TO Res.Length-1 DO
	Res.SetI(I,In.GetI(I)*Mag);
END_FOR

END_FUNCTION

// POUs/Array2DStaticMatrix
(*
Derived Matrix FB that wraps a provided 2D array of LREALS into an invariantly sized matrix
*)
{attribute 'reflection'}
{attribute 'no_assign'}
FUNCTION_BLOCK Array2DStaticMatrix EXTENDS StaticMatrix
VAR_INPUT
END_VAR
VAR_OUTPUT
END_VAR
VAR
	R0 : DINT;
	C0 : DINT;
END_VAR
VAR_IN_OUT
	Data : ARRAY[*,*] OF LREAL;
END_VAR

R0 := LOWER_BOUND(Data,1);
C0 := LOWER_BOUND(Data,2);
Init_(Array2D_Rows(Data),Array2D_Cols(Data));

//Gets the value of the element in this matrix at the supplied location as if the elements were stored in a 1D row-major array
//:Prerequisites:
// - 0 <= I < Rows*Cols
// - Matrix is not empty
//If the supplied index is out of bounds the value 0 is returned and a warning is generated in the Error List
METHOD PUBLIC GetI : LREAL//The value of the element at the specified index, or 0 if an invalid index is supplied
VAR_INPUT
	I : UINT;//The index of the element which should have its value returned
END_VAR
VAR
	Ri : UINT;
	Ci : UINT;
END_VAR
IF IsEmpty THEN
	GetI := 0.0;
	LogWarning('%s: Attempted I access of uninitialized Matrix');
ELSE
	//unwrap back into 2D
	IC2RC(I,Cols,Row => Ri,Col => Ci);
	IF Ri <0 OR Ri >= Rows OR Ci < 0 OR Ci >= Cols THEN
		GetI := 0.0;
		LogWarning('%s: Attempted I access outside of bounds of array');
	ELSE
		//add lower bound offset before fetching from array
		GetI := Data[R0+Ri,C0+Ci];
	END_IF
END_IF
END_METHOD

//Sets the element specified by the supplied index to the suppleid value, assuming the data of the matrix is stored in a 1D row-major array
//:Prerequisites: - 0 <= I < Rows*Cols
METHOD PUBLIC SetI : BOOL//TRUE if the specified index is valid and the data is copied. FLASE otherwise
VAR_INPUT
	I : UINT;//The index specifying which element should be modified
	Val : LREAL;//The value copied to the corresponding element
END_VAR
VAR
	Ri : UINT;
	Ci : UINT;
END_VAR
IF IsEmpty THEN
	SetI := FALSE;
	LogWarning('%s: Attempt to set data using I access when data is not initialized');
ELSE
	//unwrap back into 2D
	IC2RC(I,Cols,Row => Ri,Col => Ci);
	IF Ri <0 OR Ri >= Rows OR Ci < 0 OR Ci >= Cols THEN
		SetI := FALSE;
		LogWarning('%s: Attempted I access outside of bounds of array');
	ELSE
		SetI := TRUE;
		Data[R0+Ri,C0+Ci] := Val;
	END_IF
END_IF
END_METHOD

END_FUNCTION_BLOCK

// POUs/ExternalStaticMatrix
{attribute 'reflection'}
{attribute 'no_assign'}
FUNCTION_BLOCK ExternalStaticMatrix EXTENDS StaticMatrix
VAR_INPUT
END_VAR
VAR_OUTPUT
END_VAR
VAR
	Length_ : UINT;
	Data : POINTER TO LREAL;
END_VAR

METHOD PUBLIC Init
VAR_INPUT
	Buffer : POINTER TO LREAL;//must be at least length of Rows * cols!
	RowCount : UINT;
	ColCount : UINT;
END_VAR
Init_(RowCount,ColCount);
Data := BUFFER;
END_METHOD

//Gets the value of the element in this matrix at the supplied location as if the elements were stored in a 1D row-major array
//:Prerequisites:
// - I < Rows*Cols
// - Matrix is not empty
//If the supplied index is out of bounds the value 0 is returned and a warning is generated in the Error List
METHOD PUBLIC GetI : LREAL//The value of the element at the specified index, or 0 if an invalid index is supplied
VAR_INPUT
	I : UINT;//The index of the element which should have its value returned
END_VAR
IF Data = 0 THEN
	GetI := 0.0;
	LogWarning('%s: Attempted I access of uninitialized Matrix');
ELSIF I >= Length THEN
	GetI := 0.0;
	LogWarning('%s: Attempted I access of out-of-bounds Matrix data');
ELSE
	GetI := Data[I];
END_IF
END_METHOD

//Sets the element specified by the supplied index to the suppleid value, assuming the data of the matrix is stored in a 1D row-major array
//:Prerequisites: - I < Rows*Cols
METHOD PUBLIC SetI : BOOL//TRUE if the specified index is valid and the data is copied. FLASE otherwise
VAR_INPUT
	I : UINT;//The index specifying which element should be modified
	Val : LREAL;//The value copied to the corresponding element
END_VAR
IF Data = 0 THEN
	SetI := FALSE;
	LogWarning('%s: Attempt to set data using I access when data is not initialized');
ELSIF I >= Length THEN
	SetI := FALSE;
	LogWarning('%s: Attempt to set data using I access when I is out of bounds');
ELSE
	SetI := TRUE;
	Data[I] := Val;
END_IF
END_METHOD

END_FUNCTION_BLOCK
